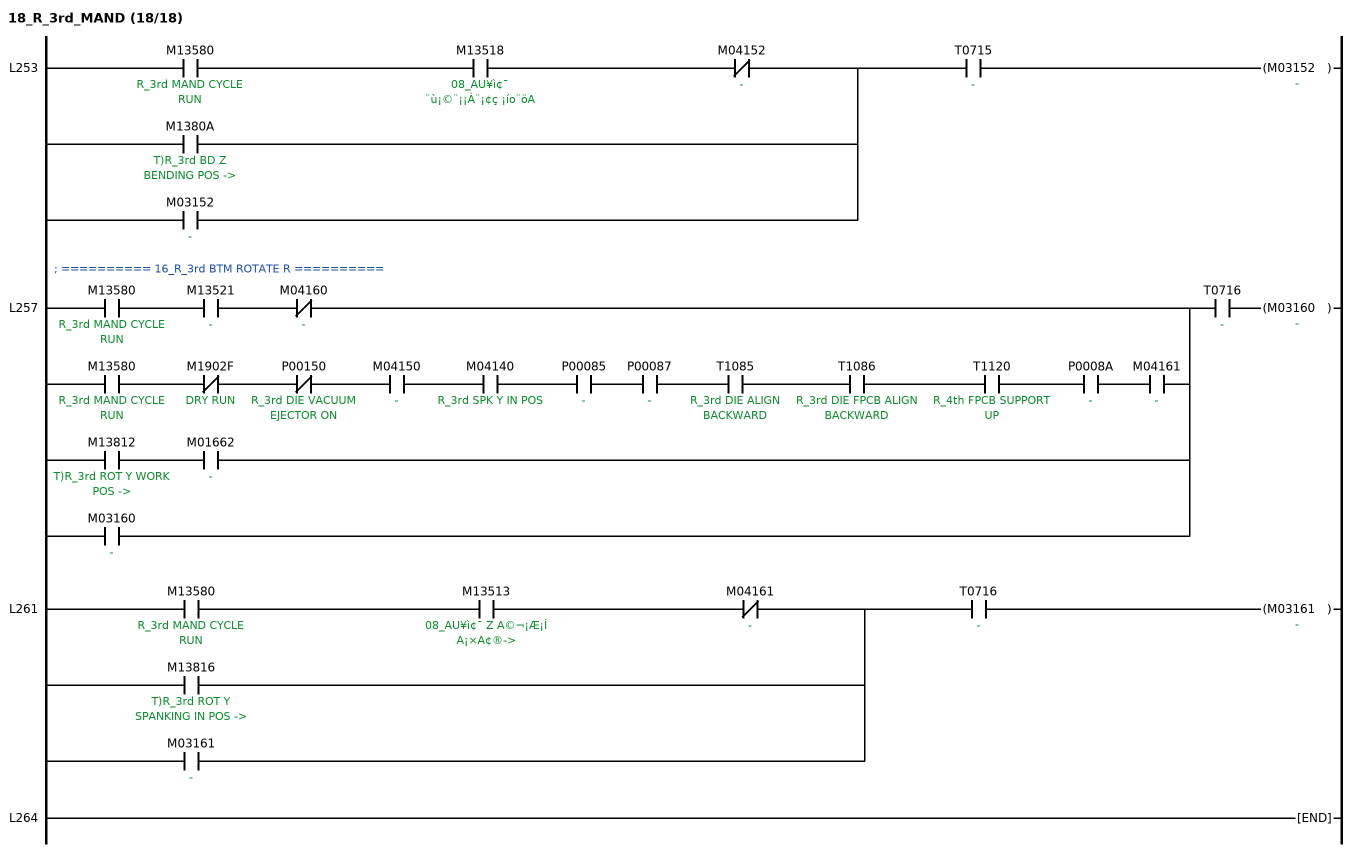
[picture p168: 18_R_3rd_MAND rungs L253-L264]
; L253
LOAD      M13580	// R_3rd MAND CYCLE RUN
AND       M13518	// 08_AU¥ì¢¯ ¨ù¡©¨¡¡À¨¡¢ç ¡ío¨öA
AND NOT   M04152	// -
OR        M1380A	// T)R_3rd BD Z BENDING POS ->
OR        M03152	// -
AND       T0715	// -
OUT       M03152	// -
// ========== 16_R_3rd BTM ROTATE R ==========
; L257
LOAD      M13580	// R_3rd MAND CYCLE RUN
AND       M13521	// -
AND NOT   M04160	// -
LOAD      M13580	// R_3rd MAND CYCLE RUN
AND NOT   M1902F	// DRY RUN
AND NOT   P00150	// R_3rd DIE VACUUM EJECTOR ON
AND       M04150	// -
AND       M04140	// R_3rd SPK Y IN POS
AND       P00085	// -
AND       P00087	// -
AND       T1085	// R_3rd DIE ALIGN BACKWARD
AND       T1086	// R_3rd DIE FPCB ALIGN BACKWARD
AND       T1120	// R_4th FPCB SUPPORT UP
AND       P0008A	// -
AND       M04161	// -
OR LOAD
LOAD      M13812	// T)R_3rd ROT Y WORK POS ->
AND       M01662	// -
OR LOAD
OR        M03160	// -
AND       T0716	// -
OUT       M03160	// -
; L261
LOAD      M13580	// R_3rd MAND CYCLE RUN
AND       M13513	// 08_AU¥ì¢¯ Z A©¬¡Æ¡Ì A¡×A¢®->
AND NOT   M04161	// -
OR        M13816	// T)R_3rd ROT Y SPANKING IN POS ->
OR        M03161	// -
AND       T0716	// -
OUT       M03161	// -
; L264
END

PROGRAM 19_R_TOOL (task: ¨ö¨¬A¥ì CA¡¤I¡¾¡¿¡¤¡Í)

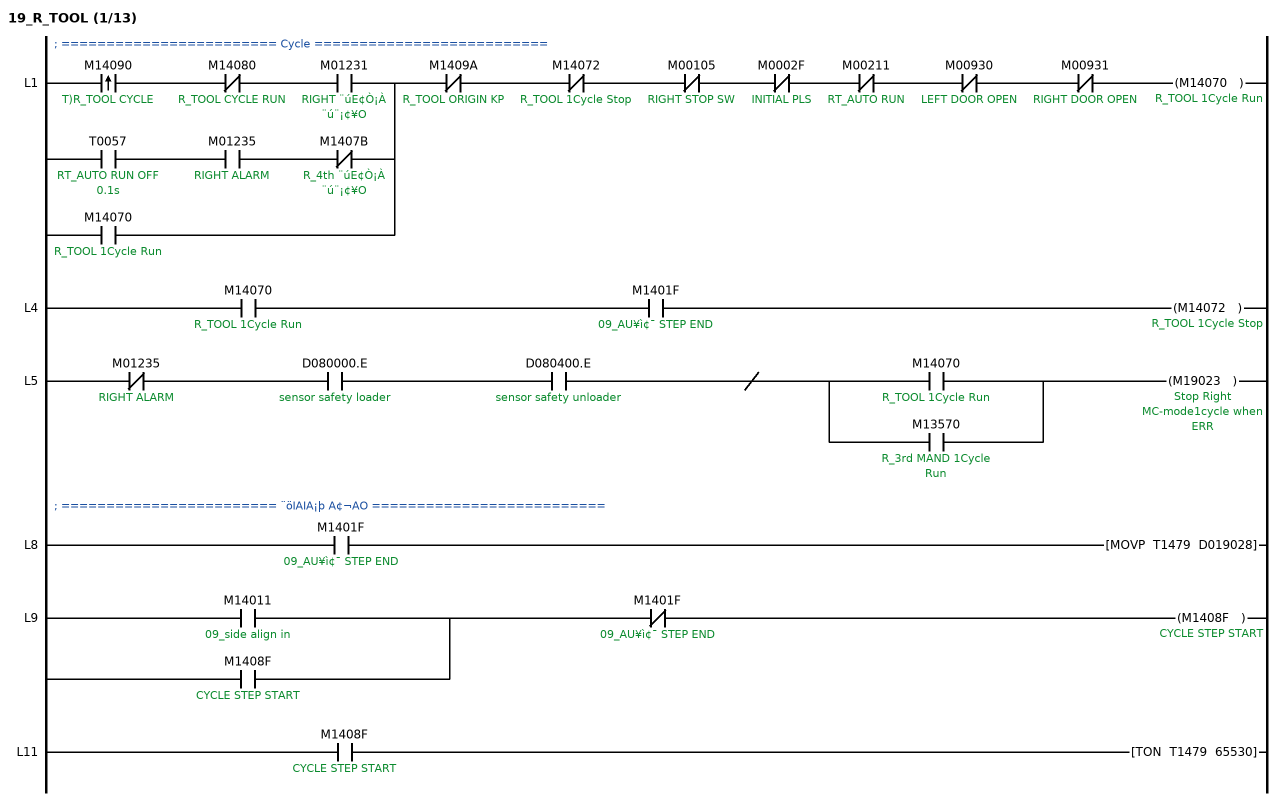
// ======================== Cycle ==========================
; L1
LOADP     M14090	// T)R_TOOL CYCLE
AND NOT   M14080	// R_TOOL CYCLE RUN
AND       M01231	// RIGHT ¨úE¢Ò¡À ¨ú¨¡¢¥O
LOAD      T0057	// RT_AUTO RUN OFF 0.1s
AND       M01235	// RIGHT ALARM
AND NOT   M1407B	// R_4th ¨úE¢Ò¡À ¨ú¨¡¢¥O
OR LOAD
OR        M14070	// R_TOOL 1Cycle Run
AND NOT   M1409A	// R_TOOL ORIGIN KP
AND NOT   M14072	// R_TOOL 1Cycle Stop
AND NOT   M00105	// RIGHT STOP SW
AND NOT   M0002F	// INITIAL PLS
AND NOT   M00211	// RT_AUTO RUN
AND NOT   M00930	// LEFT DOOR OPEN
AND NOT   M00931	// RIGHT DOOR OPEN
OUT       M14070	// R_TOOL 1Cycle Run
; L4
LOAD      M14070	// R_TOOL 1Cycle Run
AND       M1401F	// 09_AU¥ì¢¯ STEP END
OUT       M14072	// R_TOOL 1Cycle Stop
; L5
LOAD NOT  M01235	// RIGHT ALARM
AND       D080000.E	// sensor safety loader
AND       D080400.E	// sensor safety unloader
NOT
LOAD      M14070	// R_TOOL 1Cycle Run
OR        M13570	// R_3rd MAND 1Cycle Run
AND LOAD
OUT       M19023	// Stop Right MC-mode1cycle when ERR
// ======================== ¨öIAIA¡þ A¢¬AO ==========================
; L8
LOAD      M1401F	// 09_AU¥ì¢¯ STEP END
MOVP      T1479 D019028
; L9
LOAD      M14011	// 09_side align in
OR        M1408F	// CYCLE STEP START
AND NOT   M1401F	// 09_AU¥ì¢¯ STEP END
OUT       M1408F	// CYCLE STEP START
; L11
LOAD      M1408F	// CYCLE STEP START
TON       T1479 65530

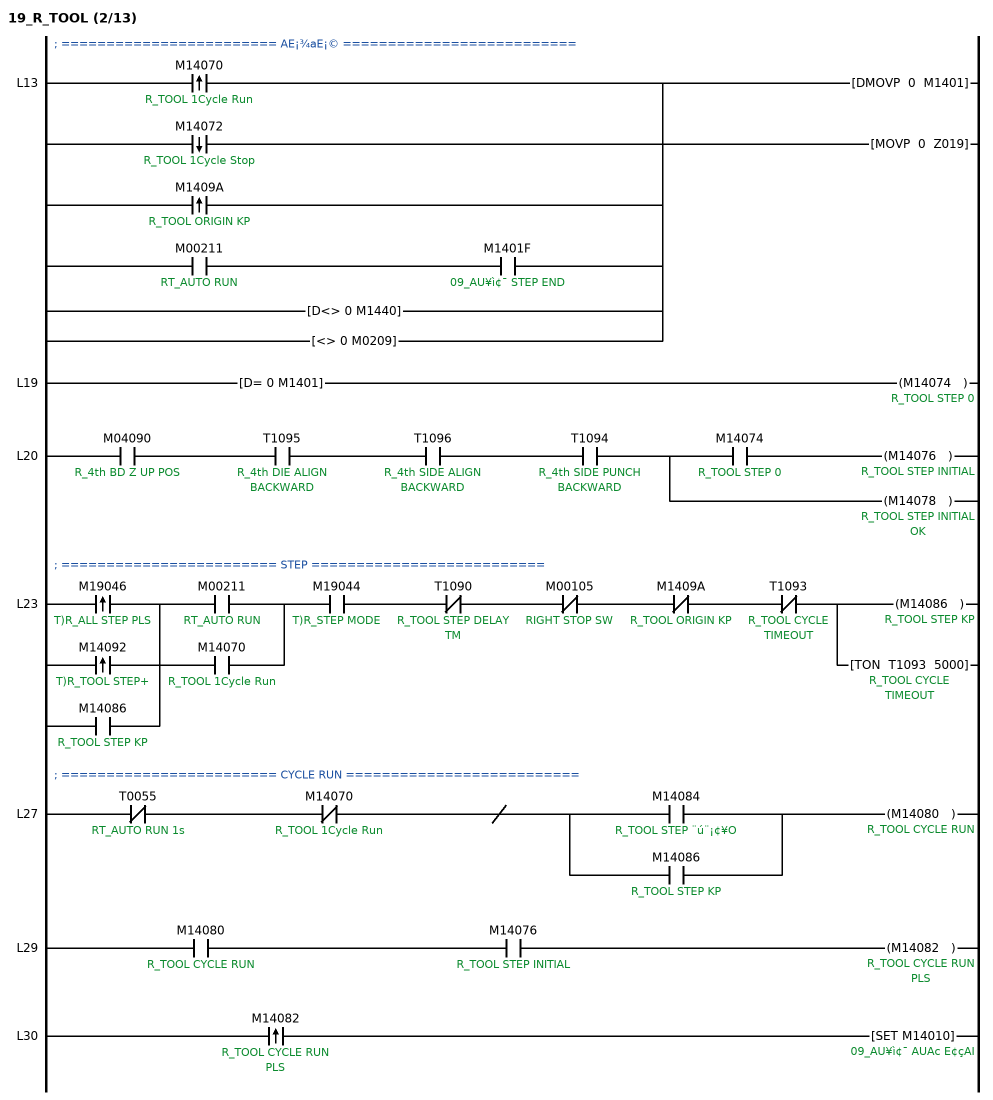
// ======================== AE¡¾aE¡© ==========================
; L13
LOADP     M14070	// R_TOOL 1Cycle Run
ORN       M14072	// R_TOOL 1Cycle Stop
ORP       M1409A	// R_TOOL ORIGIN KP
LOAD      M00211	// RT_AUTO RUN
AND       M1401F	// 09_AU¥ì¢¯ STEP END
OR LOAD
ORD<>     0 M1440
OR<>      0 M0209
DMOVP     0 M1401
MOVP      0 Z019
; L19
LOADD=    0 M1401
OUT       M14074	// R_TOOL STEP 0
; L20
LOAD      M04090	// R_4th BD Z UP POS
AND       T1095	// R_4th DIE ALIGN BACKWARD
AND       T1096	// R_4th SIDE ALIGN BACKWARD
AND       T1094	// R_4th SIDE PUNCH BACKWARD
MPUSH
AND       M14074	// R_TOOL STEP 0
OUT       M14076	// R_TOOL STEP INITIAL
MPOP
OUT       M14078	// R_TOOL STEP INITIAL OK
// ======================== STEP ==========================
; L23
LOADP     M19046	// T)R_ALL STEP PLS
ORP       M14092	// T)R_TOOL STEP+
OR        M14086	// R_TOOL STEP KP
LOAD      M00211	// RT_AUTO RUN
OR        M14070	// R_TOOL 1Cycle Run
AND LOAD
AND       M19044	// T)R_STEP MODE
AND NOT   T1090	// R_TOOL STEP DELAY TM
AND NOT   M00105	// RIGHT STOP SW
AND NOT   M1409A	// R_TOOL ORIGIN KP
AND NOT   T1093	// R_TOOL CYCLE TIMEOUT
OUT       M14086	// R_TOOL STEP KP
TON       T1093 5000	// R_TOOL CYCLE TIMEOUT
// ======================== CYCLE RUN ==========================
; L27
LOAD NOT  T0055	// RT_AUTO RUN 1s
AND NOT   M14070	// R_TOOL 1Cycle Run
NOT
LOAD      M14084	// R_TOOL STEP ¨ú¨¡¢¥O
OR        M14086	// R_TOOL STEP KP
AND LOAD
OUT       M14080	// R_TOOL CYCLE RUN
; L29
LOAD      M14080	// R_TOOL CYCLE RUN
AND       M14076	// R_TOOL STEP INITIAL
OUT       M14082	// R_TOOL CYCLE RUN PLS
; L30
LOADP     M14082	// R_TOOL CYCLE RUN PLS
SET       M14010	// 09_AU¥ì¢¯ AUAc E¢çAI

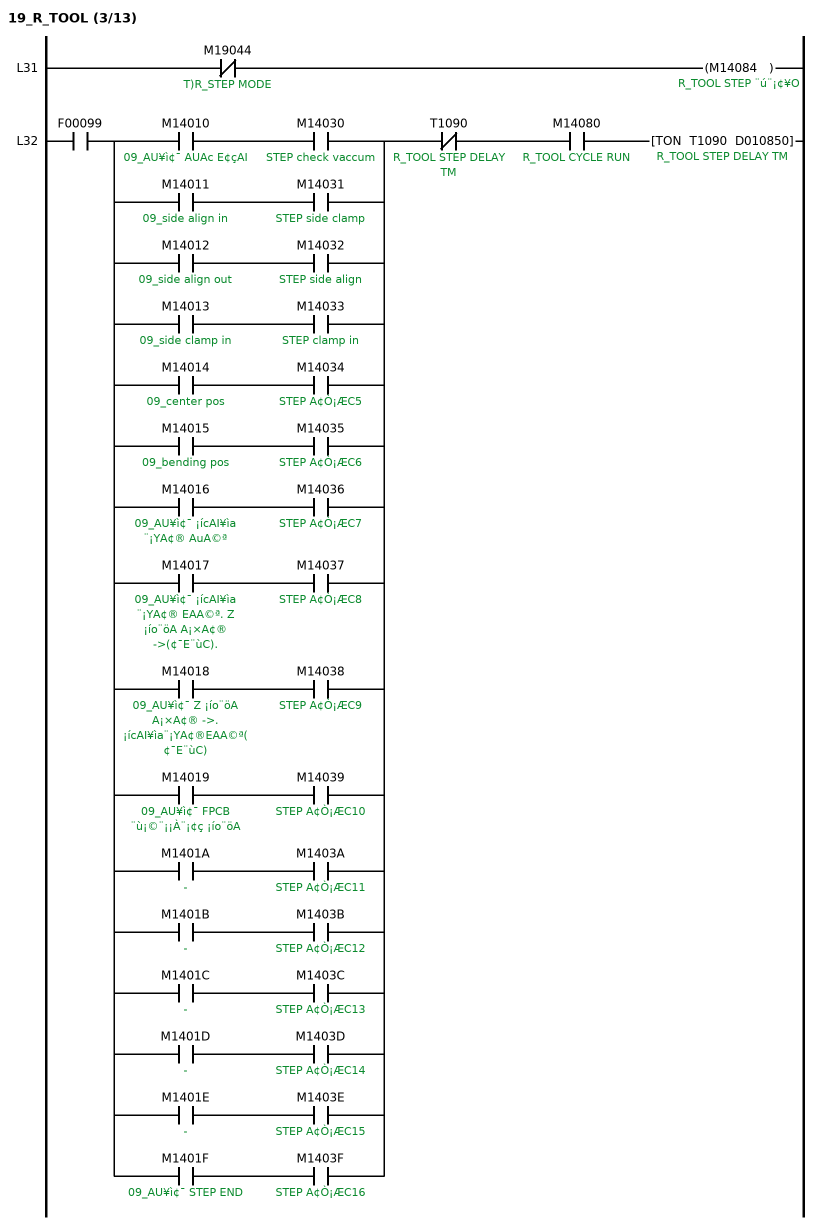
; L31
LOAD NOT  M19044	// T)R_STEP MODE
OUT       M14084	// R_TOOL STEP ¨ú¨¡¢¥O
; L32
LOAD      F00099
LOAD      M14010	// 09_AU¥ì¢¯ AUAc E¢çAI
AND       M14030	// STEP check vaccum
LOAD      M14011	// 09_side align in
AND       M14031	// STEP side clamp
OR LOAD
LOAD      M14012	// 09_side align out
AND       M14032	// STEP side align
OR LOAD
LOAD      M14013	// 09_side clamp in
AND       M14033	// STEP clamp in
OR LOAD
LOAD      M14014	// 09_center pos
AND       M14034	// STEP A¢Ò¡ÆC5
OR LOAD
LOAD      M14015	// 09_bending pos
AND       M14035	// STEP A¢Ò¡ÆC6
OR LOAD
LOAD      M14016	// 09_AU¥ì¢¯ ¡ícAI¥ìa ¨¡YA¢® AuA©ª
AND       M14036	// STEP A¢Ò¡ÆC7
OR LOAD
LOAD      M14017	// 09_AU¥ì¢¯ ¡ícAI¥ìa ¨¡YA¢® EAA©ª. Z ¡ío¨öA A¡×A¢® ->(¢¯E¨ùC).
AND       M14037	// STEP A¢Ò¡ÆC8
OR LOAD
LOAD      M14018	// 09_AU¥ì¢¯ Z ¡ío¨öA A¡×A¢® ->. ¡ícAI¥ìa¨¡YA¢®EAA©ª(¢¯E¨ùC)
AND       M14038	// STEP A¢Ò¡ÆC9
OR LOAD
LOAD      M14019	// 09_AU¥ì¢¯ FPCB ¨ù¡©¨¡¡À¨¡¢ç ¡ío¨öA
AND       M14039	// STEP A¢Ò¡ÆC10
OR LOAD
LOAD      M1401A	// -
AND       M1403A	// STEP A¢Ò¡ÆC11
OR LOAD
LOAD      M1401B	// -
AND       M1403B	// STEP A¢Ò¡ÆC12
OR LOAD
LOAD      M1401C	// -
AND       M1403C	// STEP A¢Ò¡ÆC13
OR LOAD
LOAD      M1401D	// -
AND       M1403D	// STEP A¢Ò¡ÆC14
OR LOAD
LOAD      M1401E	// -
AND       M1403E	// STEP A¢Ò¡ÆC15
OR LOAD
LOAD      M1401F	// 09_AU¥ì¢¯ STEP END
AND       M1403F	// STEP A¢Ò¡ÆC16
OR LOAD
AND LOAD
AND NOT   T1090	// R_TOOL STEP DELAY TM
AND       M14080	// R_TOOL CYCLE RUN
TON       T1090 D010850	// R_TOOL STEP DELAY TM

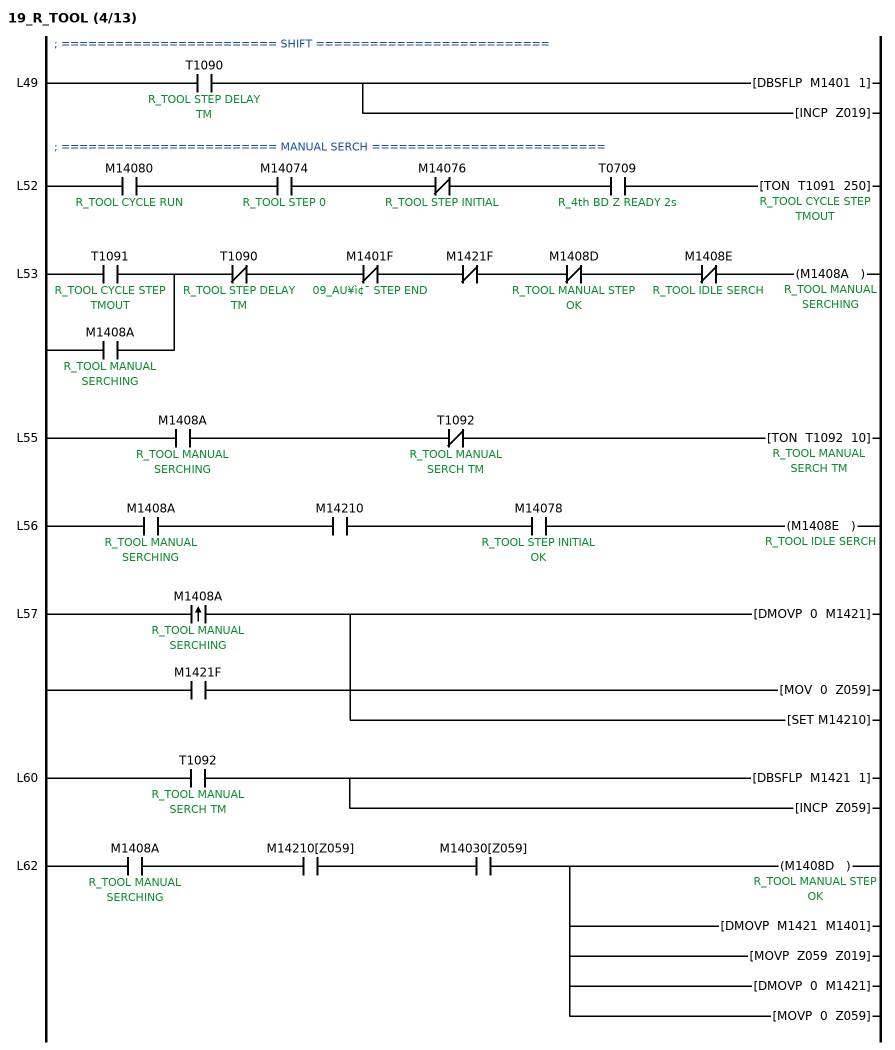
// ======================== SHIFT ==========================
; L49
LOAD      T1090	// R_TOOL STEP DELAY TM
DBSFLP    M1401 1
INCP      Z019
// ======================== MANUAL SERCH ==========================
; L52
LOAD      M14080	// R_TOOL CYCLE RUN
AND       M14074	// R_TOOL STEP 0
AND NOT   M14076	// R_TOOL STEP INITIAL
AND       T0709	// R_4th BD Z READY 2s
TON       T1091 250	// R_TOOL CYCLE STEP TMOUT
; L53
LOAD      T1091	// R_TOOL CYCLE STEP TMOUT
OR        M1408A	// R_TOOL MANUAL SERCHING
AND NOT   T1090	// R_TOOL STEP DELAY TM
AND NOT   M1401F	// 09_AU¥ì¢¯ STEP END
AND NOT   M1421F
AND NOT   M1408D	// R_TOOL MANUAL STEP OK
AND NOT   M1408E	// R_TOOL IDLE SERCH
OUT       M1408A	// R_TOOL MANUAL SERCHING
; L55
LOAD      M1408A	// R_TOOL MANUAL SERCHING
AND NOT   T1092	// R_TOOL MANUAL SERCH TM
TON       T1092 10	// R_TOOL MANUAL SERCH TM
; L56
LOAD      M1408A	// R_TOOL MANUAL SERCHING
AND       M14210
AND       M14078	// R_TOOL STEP INITIAL OK
OUT       M1408E	// R_TOOL IDLE SERCH
; L57
LOADP     M1408A	// R_TOOL MANUAL SERCHING
OR        M1421F
DMOVP     0 M1421
MOV       0 Z059
SET       M14210
; L60
LOAD      T1092	// R_TOOL MANUAL SERCH TM
DBSFLP    M1421 1
INCP      Z059
; L62
LOAD      M1408A	// R_TOOL MANUAL SERCHING
AND       M14210[Z059]
AND       M14030[Z059]
OUT       M1408D	// R_TOOL MANUAL STEP OK
DMOVP     M1421 M1401
MOVP      Z059 Z019
DMOVP     0 M1421
MOVP      0 Z059

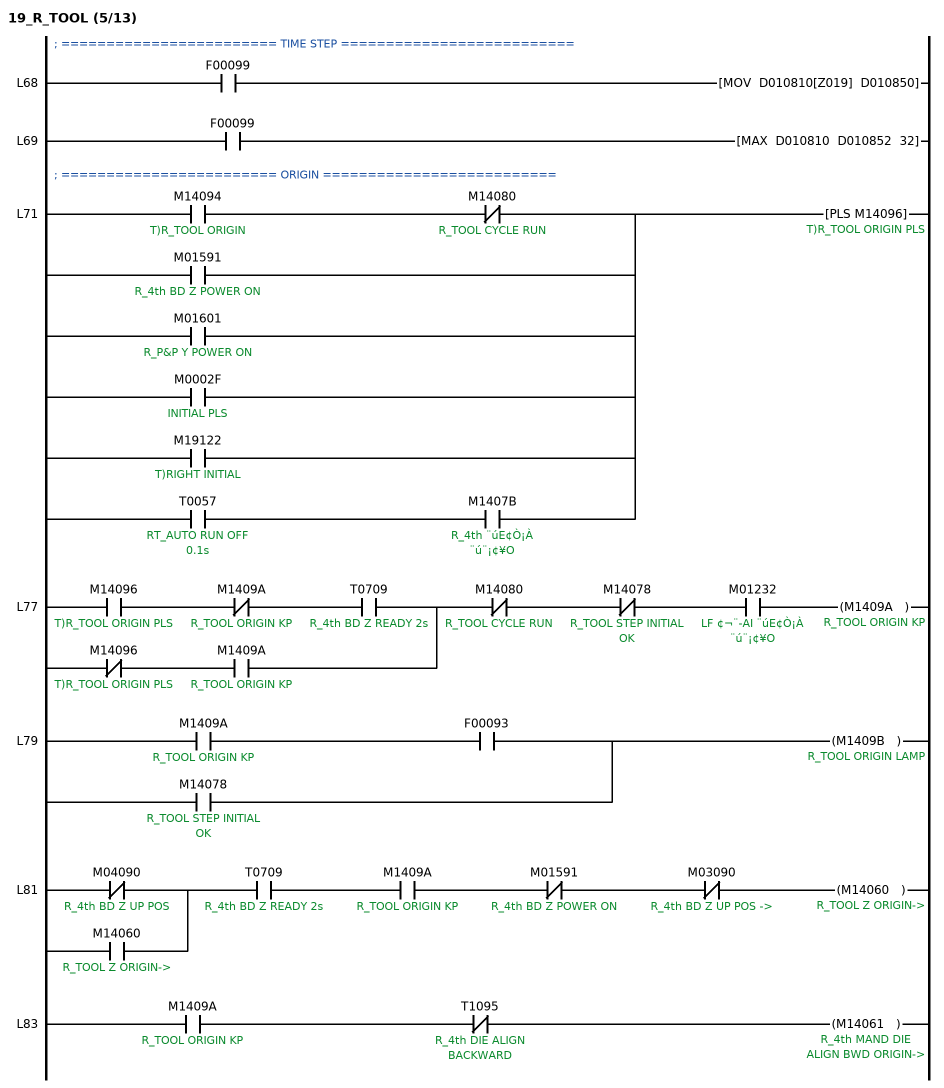
// ======================== TIME STEP ==========================
; L68
LOAD      F00099
MOV       D010810[Z019] D010850
; L69
LOAD      F00099
MAX       D010810 D010852 32
// ======================== ORIGIN ==========================
; L71
LOAD      M14094	// T)R_TOOL ORIGIN
AND NOT   M14080	// R_TOOL CYCLE RUN
OR        M01591	// R_4th BD Z POWER ON
OR        M01601	// R_P&P Y POWER ON
OR        M0002F	// INITIAL PLS
OR        M19122	// T)RIGHT INITIAL
LOAD      T0057	// RT_AUTO RUN OFF 0.1s
AND       M1407B	// R_4th ¨úE¢Ò¡À ¨ú¨¡¢¥O
OR LOAD
OUTP      M14096	// T)R_TOOL ORIGIN PLS
; L77
LOAD      M14096	// T)R_TOOL ORIGIN PLS
AND NOT   M1409A	// R_TOOL ORIGIN KP
AND       T0709	// R_4th BD Z READY 2s
LOAD NOT  M14096	// T)R_TOOL ORIGIN PLS
AND       M1409A	// R_TOOL ORIGIN KP
OR LOAD
AND NOT   M14080	// R_TOOL CYCLE RUN
AND NOT   M14078	// R_TOOL STEP INITIAL OK
AND       M01232	// LF ¢¬¨­AI ¨úE¢Ò¡À ¨ú¨¡¢¥O
OUT       M1409A	// R_TOOL ORIGIN KP
; L79
LOAD      M1409A	// R_TOOL ORIGIN KP
AND       F00093
OR        M14078	// R_TOOL STEP INITIAL OK
OUT       M1409B	// R_TOOL ORIGIN LAMP
; L81
LOAD NOT  M04090	// R_4th BD Z UP POS
OR        M14060	// R_TOOL Z ORIGIN->
AND       T0709	// R_4th BD Z READY 2s
AND       M1409A	// R_TOOL ORIGIN KP
AND NOT   M01591	// R_4th BD Z POWER ON
AND NOT   M03090	// R_4th BD Z UP POS ->
OUT       M14060	// R_TOOL Z ORIGIN->
; L83
LOAD      M1409A	// R_TOOL ORIGIN KP
AND NOT   T1095	// R_4th DIE ALIGN BACKWARD
OUT       M14061	// R_4th MAND DIE ALIGN BWD ORIGIN->

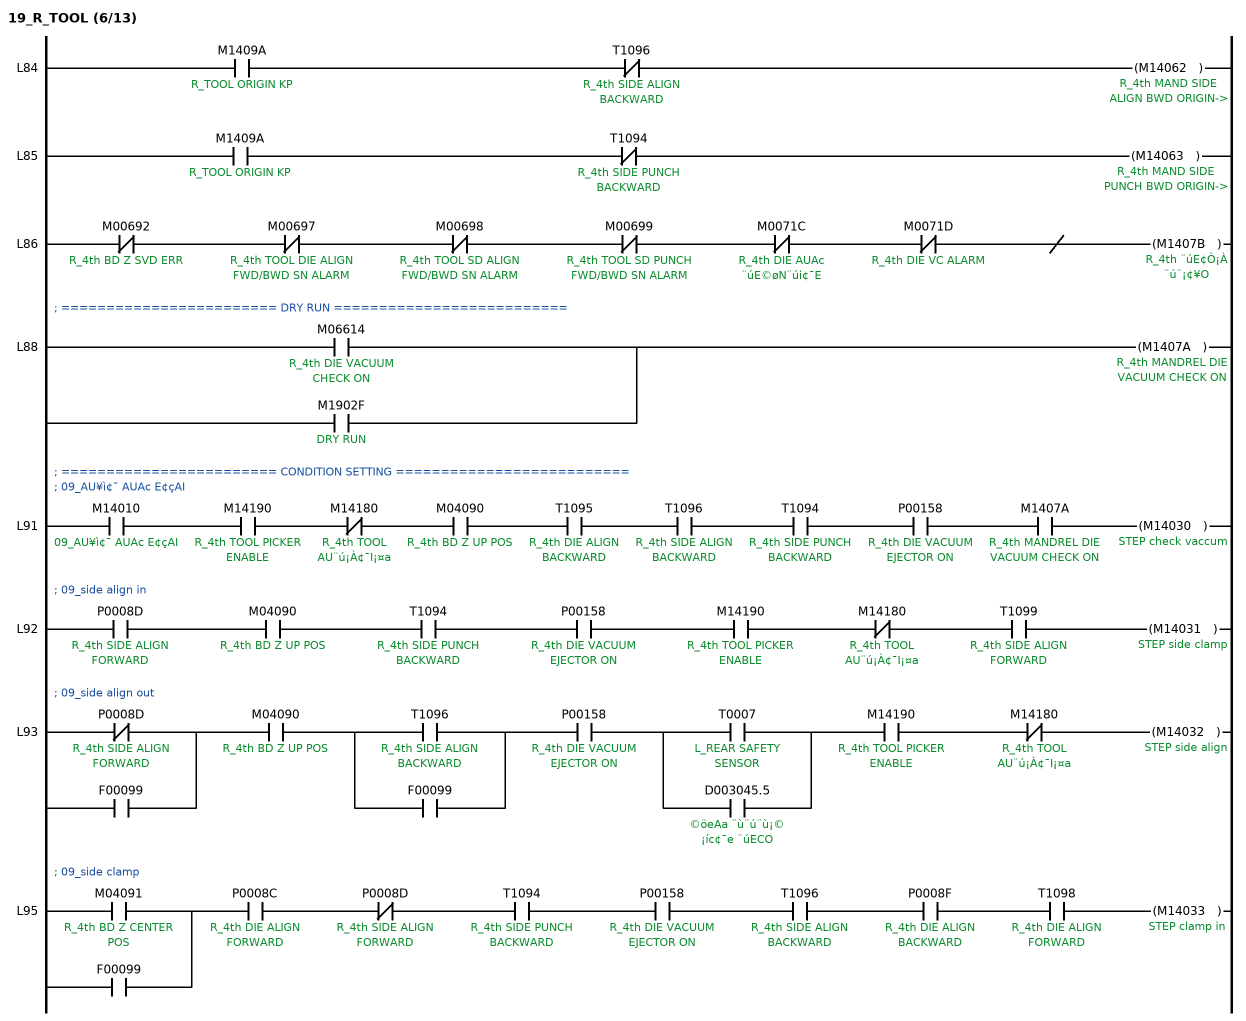
; L84
LOAD      M1409A	// R_TOOL ORIGIN KP
AND NOT   T1096	// R_4th SIDE ALIGN BACKWARD
OUT       M14062	// R_4th MAND SIDE ALIGN BWD ORIGIN->
; L85
LOAD      M1409A	// R_TOOL ORIGIN KP
AND NOT   T1094	// R_4th SIDE PUNCH BACKWARD
OUT       M14063	// R_4th MAND SIDE PUNCH BWD ORIGIN->
; L86
LOAD NOT  M00692	// R_4th BD Z SVD ERR
AND NOT   M00697	// R_4th TOOL DIE ALIGN FWD/BWD SN ALARM
AND NOT   M00698	// R_4th TOOL SD ALIGN FWD/BWD SN ALARM
AND NOT   M00699	// R_4th TOOL SD PUNCH FWD/BWD SN ALARM
AND NOT   M0071C	// R_4th DIE AUAc ¨úE©øN¨úi¢¯E
AND NOT   M0071D	// R_4th DIE VC ALARM
NOT
OUT       M1407B	// R_4th ¨úE¢Ò¡À ¨ú¨¡¢¥O
// ======================== DRY RUN ==========================
; L88
LOAD      M06614	// R_4th DIE VACUUM CHECK ON
OR        M1902F	// DRY RUN
OUT       M1407A	// R_4th MANDREL DIE VACUUM CHECK ON
// ======================== CONDITION SETTING ==========================
; L91
LOAD      M14010	// 09_AU¥ì¢¯ AUAc E¢çAI
AND       M14190	// R_4th TOOL PICKER ENABLE
AND NOT   M14180	// R_4th TOOL AU¨ú¡À¢¯I¡¤a
AND       M04090	// R_4th BD Z UP POS
AND       T1095	// R_4th DIE ALIGN BACKWARD
AND       T1096	// R_4th SIDE ALIGN BACKWARD
AND       T1094	// R_4th SIDE PUNCH BACKWARD
AND       P00158	// R_4th DIE VACUUM EJECTOR ON
AND       M1407A	// R_4th MANDREL DIE VACUUM CHECK ON
OUT       M14030	// STEP check vaccum
// output comment: 09_AU¥ì¢¯ AUAc E¢çAI
; L92
LOAD      P0008D	// R_4th SIDE ALIGN FORWARD
AND       M04090	// R_4th BD Z UP POS
AND       T1094	// R_4th SIDE PUNCH BACKWARD
AND       P00158	// R_4th DIE VACUUM EJECTOR ON
AND       M14190	// R_4th TOOL PICKER ENABLE
AND NOT   M14180	// R_4th TOOL AU¨ú¡À¢¯I¡¤a
AND       T1099	// R_4th SIDE ALIGN FORWARD
OUT       M14031	// STEP side clamp
// output comment: 09_side align in
; L93
LOAD NOT  P0008D	// R_4th SIDE ALIGN FORWARD
OR        F00099
AND       M04090	// R_4th BD Z UP POS
LOAD      T1096	// R_4th SIDE ALIGN BACKWARD
OR        F00099
AND LOAD
AND       P00158	// R_4th DIE VACUUM EJECTOR ON
LOAD      T0007	// L_REAR SAFETY SENSOR
OR        D003045.5	// ©öeAa ¨ù¨ú¨ù¡© ¡íc¢¯e ¨úECO
AND LOAD
AND       M14190	// R_4th TOOL PICKER ENABLE
AND NOT   M14180	// R_4th TOOL AU¨ú¡À¢¯I¡¤a
OUT       M14032	// STEP side align
// output comment: 09_side align out
; L95
LOAD      M04091	// R_4th BD Z CENTER POS
OR        F00099
AND       P0008C	// R_4th DIE ALIGN FORWARD
AND NOT   P0008D	// R_4th SIDE ALIGN FORWARD
AND       T1094	// R_4th SIDE PUNCH BACKWARD
AND       P00158	// R_4th DIE VACUUM EJECTOR ON
AND       T1096	// R_4th SIDE ALIGN BACKWARD
AND       P0008F	// R_4th DIE ALIGN BACKWARD
AND       T1098	// R_4th DIE ALIGN FORWARD
OUT       M14033	// STEP clamp in
// output comment: 09_side clamp

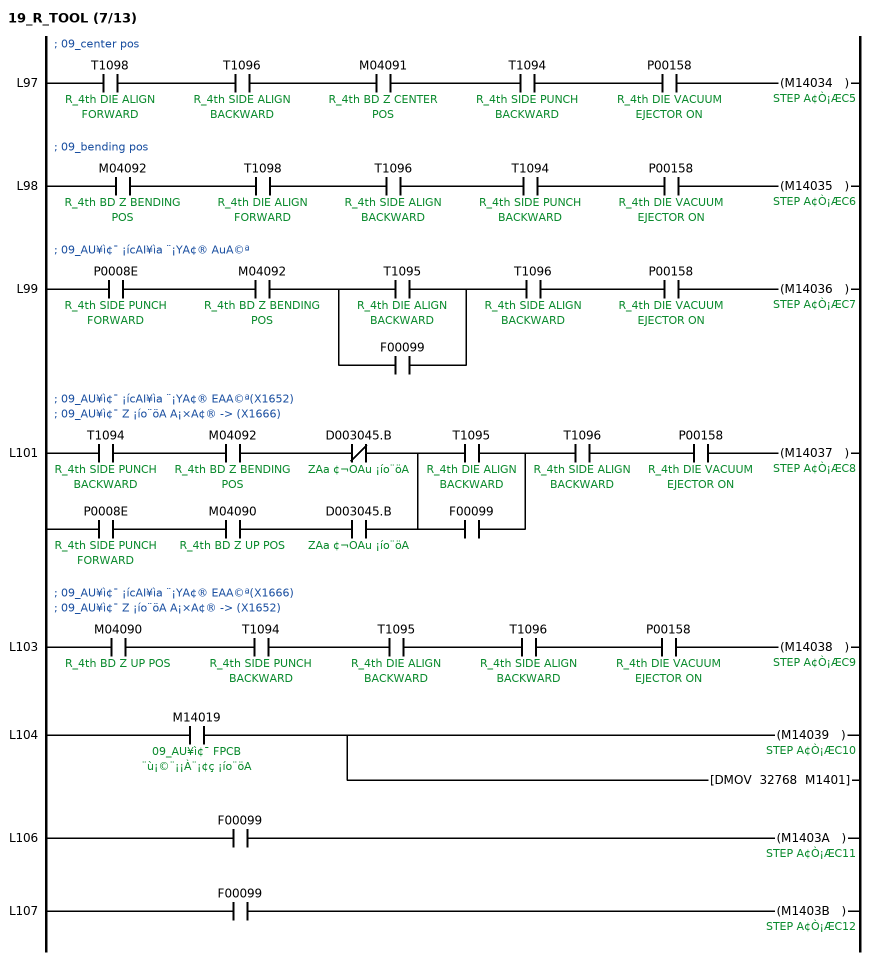
; L97
LOAD      T1098	// R_4th DIE ALIGN FORWARD
AND       T1096	// R_4th SIDE ALIGN BACKWARD
AND       M04091	// R_4th BD Z CENTER POS
AND       T1094	// R_4th SIDE PUNCH BACKWARD
AND       P00158	// R_4th DIE VACUUM EJECTOR ON
OUT       M14034	// STEP A¢Ò¡ÆC5
// output comment: 09_center pos
; L98
LOAD      M04092	// R_4th BD Z BENDING POS
AND       T1098	// R_4th DIE ALIGN FORWARD
AND       T1096	// R_4th SIDE ALIGN BACKWARD
AND       T1094	// R_4th SIDE PUNCH BACKWARD
AND       P00158	// R_4th DIE VACUUM EJECTOR ON
OUT       M14035	// STEP A¢Ò¡ÆC6
// output comment: 09_bending pos
; L99
LOAD      P0008E	// R_4th SIDE PUNCH FORWARD
AND       M04092	// R_4th BD Z BENDING POS
LOAD      T1095	// R_4th DIE ALIGN BACKWARD
OR        F00099
AND LOAD
AND       T1096	// R_4th SIDE ALIGN BACKWARD
AND       P00158	// R_4th DIE VACUUM EJECTOR ON
OUT       M14036	// STEP A¢Ò¡ÆC7
// output comment: 09_AU¥ì¢¯ ¡ícAI¥ìa ¨¡YA¢® AuA©ª
; L101
LOAD      T1094	// R_4th SIDE PUNCH BACKWARD
AND       M04092	// R_4th BD Z BENDING POS
AND NOT   D003045.B	// ZAa ¢¬OAu ¡ío¨öA
LOAD      P0008E	// R_4th SIDE PUNCH FORWARD
AND       M04090	// R_4th BD Z UP POS
AND       D003045.B	// ZAa ¢¬OAu ¡ío¨öA
OR LOAD
LOAD      T1095	// R_4th DIE ALIGN BACKWARD
OR        F00099
AND LOAD
AND       T1096	// R_4th SIDE ALIGN BACKWARD
AND       P00158	// R_4th DIE VACUUM EJECTOR ON
OUT       M14037	// STEP A¢Ò¡ÆC8
// output comment: 09_AU¥ì¢¯ ¡ícAI¥ìa ¨¡YA¢® EAA©ª(X1652) 09_AU¥ì¢¯ Z ¡ío¨öA A¡×A¢® -> (X1666)
; L103
LOAD      M04090	// R_4th BD Z UP POS
AND       T1094	// R_4th SIDE PUNCH BACKWARD
AND       T1095	// R_4th DIE ALIGN BACKWARD
AND       T1096	// R_4th SIDE ALIGN BACKWARD
AND       P00158	// R_4th DIE VACUUM EJECTOR ON
OUT       M14038	// STEP A¢Ò¡ÆC9
// output comment: 09_AU¥ì¢¯ ¡ícAI¥ìa ¨¡YA¢® EAA©ª(X1666) 09_AU¥ì¢¯ Z ¡ío¨öA A¡×A¢® -> (X1652)
; L104
LOAD      M14019	// 09_AU¥ì¢¯ FPCB ¨ù¡©¨¡¡À¨¡¢ç ¡ío¨öA
OUT       M14039	// STEP A¢Ò¡ÆC10
DMOV      32768 M1401
; L106
LOAD      F00099
OUT       M1403A	// STEP A¢Ò¡ÆC11
; L107
LOAD      F00099
OUT       M1403B	// STEP A¢Ò¡ÆC12

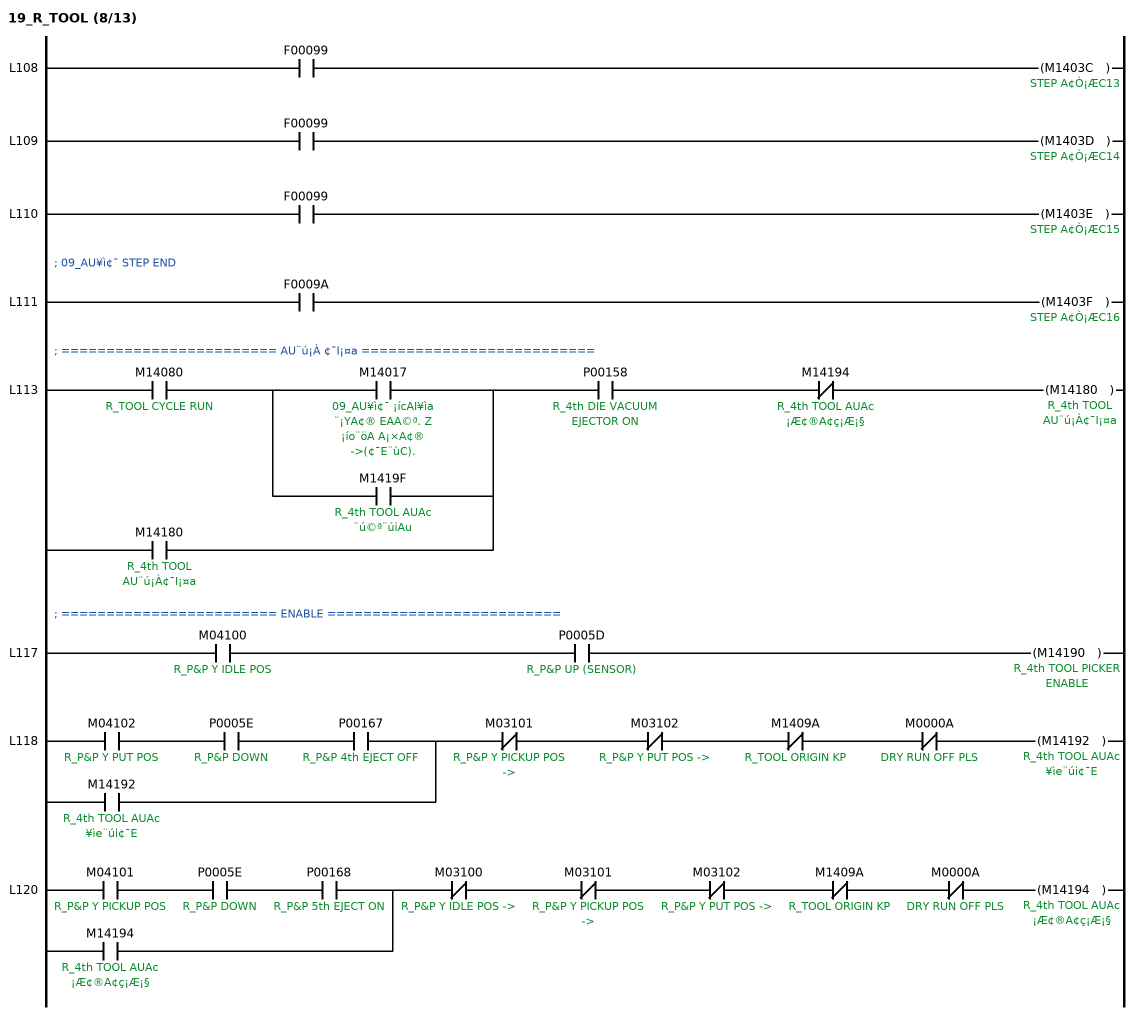
; L108
LOAD      F00099
OUT       M1403C	// STEP A¢Ò¡ÆC13
; L109
LOAD      F00099
OUT       M1403D	// STEP A¢Ò¡ÆC14
; L110
LOAD      F00099
OUT       M1403E	// STEP A¢Ò¡ÆC15
; L111
LOAD      F0009A
OUT       M1403F	// STEP A¢Ò¡ÆC16
// output comment: 09_AU¥ì¢¯ STEP END
// ======================== AU¨ú¡À ¢¯I¡¤a ==========================
; L113
LOAD      M14080	// R_TOOL CYCLE RUN
LOAD      M14017	// 09_AU¥ì¢¯ ¡ícAI¥ìa ¨¡YA¢® EAA©ª. Z ¡ío¨öA A¡×A¢® ->(¢¯E¨ùC).
OR        M1419F	// R_4th TOOL AUAc ¨ú©ª¨úiAu
AND LOAD
OR        M14180	// R_4th TOOL AU¨ú¡À¢¯I¡¤a
AND       P00158	// R_4th DIE VACUUM EJECTOR ON
AND NOT   M14194	// R_4th TOOL AUAc ¡Æ¢®A¢ç¡Æ¡§
OUT       M14180	// R_4th TOOL AU¨ú¡À¢¯I¡¤a
// ======================== ENABLE ==========================
; L117
LOAD      M04100	// R_P&P Y IDLE POS
AND       P0005D	// R_P&P UP (SENSOR)
OUT       M14190	// R_4th TOOL PICKER ENABLE
; L118
LOAD      M04102	// R_P&P Y PUT POS
AND       P0005E	// R_P&P DOWN
AND       P00167	// R_P&P 4th EJECT OFF
OR        M14192	// R_4th TOOL AUAc ¥ìe¨úi¢¯E
AND NOT   M03101	// R_P&P Y PICKUP POS ->
AND NOT   M03102	// R_P&P Y PUT POS ->
AND NOT   M1409A	// R_TOOL ORIGIN KP
AND NOT   M0000A	// DRY RUN OFF PLS
OUT       M14192	// R_4th TOOL AUAc ¥ìe¨úi¢¯E
; L120
LOAD      M04101	// R_P&P Y PICKUP POS
AND       P0005E	// R_P&P DOWN
AND       P00168	// R_P&P 5th EJECT ON
OR        M14194	// R_4th TOOL AUAc ¡Æ¢®A¢ç¡Æ¡§
AND NOT   M03100	// R_P&P Y IDLE POS ->
AND NOT   M03101	// R_P&P Y PICKUP POS ->
AND NOT   M03102	// R_P&P Y PUT POS ->
AND NOT   M1409A	// R_TOOL ORIGIN KP
AND NOT   M0000A	// DRY RUN OFF PLS
OUT       M14194	// R_4th TOOL AUAc ¡Æ¢®A¢ç¡Æ¡§

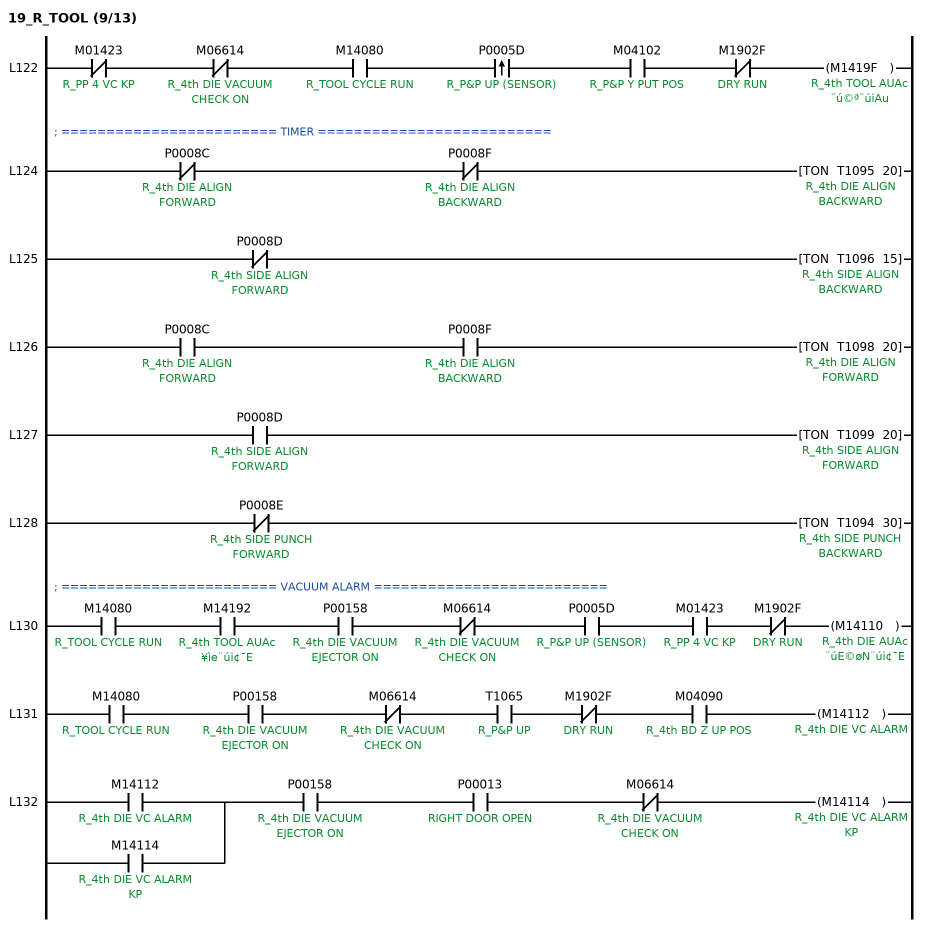
; L122
LOAD NOT  M01423	// R_PP 4 VC KP
AND NOT   M06614	// R_4th DIE VACUUM CHECK ON
AND       M14080	// R_TOOL CYCLE RUN
ANDP      P0005D	// R_P&P UP (SENSOR)
AND       M04102	// R_P&P Y PUT POS
AND NOT   M1902F	// DRY RUN
OUT       M1419F	// R_4th TOOL AUAc ¨ú©ª¨úiAu
// ======================== TIMER ==========================
; L124
LOAD NOT  P0008C	// R_4th DIE ALIGN FORWARD
AND NOT   P0008F	// R_4th DIE ALIGN BACKWARD
TON       T1095 20	// R_4th DIE ALIGN BACKWARD
; L125
LOAD NOT  P0008D	// R_4th SIDE ALIGN FORWARD
TON       T1096 15	// R_4th SIDE ALIGN BACKWARD
; L126
LOAD      P0008C	// R_4th DIE ALIGN FORWARD
AND       P0008F	// R_4th DIE ALIGN BACKWARD
TON       T1098 20	// R_4th DIE ALIGN FORWARD
; L127
LOAD      P0008D	// R_4th SIDE ALIGN FORWARD
TON       T1099 20	// R_4th SIDE ALIGN FORWARD
; L128
LOAD NOT  P0008E	// R_4th SIDE PUNCH FORWARD
TON       T1094 30	// R_4th SIDE PUNCH BACKWARD
// ======================== VACUUM ALARM ==========================
; L130
LOAD      M14080	// R_TOOL CYCLE RUN
AND       M14192	// R_4th TOOL AUAc ¥ìe¨úi¢¯E
AND       P00158	// R_4th DIE VACUUM EJECTOR ON
AND NOT   M06614	// R_4th DIE VACUUM CHECK ON
AND       P0005D	// R_P&P UP (SENSOR)
AND       M01423	// R_PP 4 VC KP
AND NOT   M1902F	// DRY RUN
OUT       M14110	// R_4th DIE AUAc ¨úE©øN¨úi¢¯E
; L131
LOAD      M14080	// R_TOOL CYCLE RUN
AND       P00158	// R_4th DIE VACUUM EJECTOR ON
AND NOT   M06614	// R_4th DIE VACUUM CHECK ON
AND       T1065	// R_P&P UP
AND NOT   M1902F	// DRY RUN
AND       M04090	// R_4th BD Z UP POS
OUT       M14112	// R_4th DIE VC ALARM
; L132
LOAD      M14112	// R_4th DIE VC ALARM
OR        M14114	// R_4th DIE VC ALARM KP
AND       P00158	// R_4th DIE VACUUM EJECTOR ON
AND       P00013	// RIGHT DOOR OPEN
AND NOT   M06614	// R_4th DIE VACUUM CHECK ON
OUT       M14114	// R_4th DIE VC ALARM KP

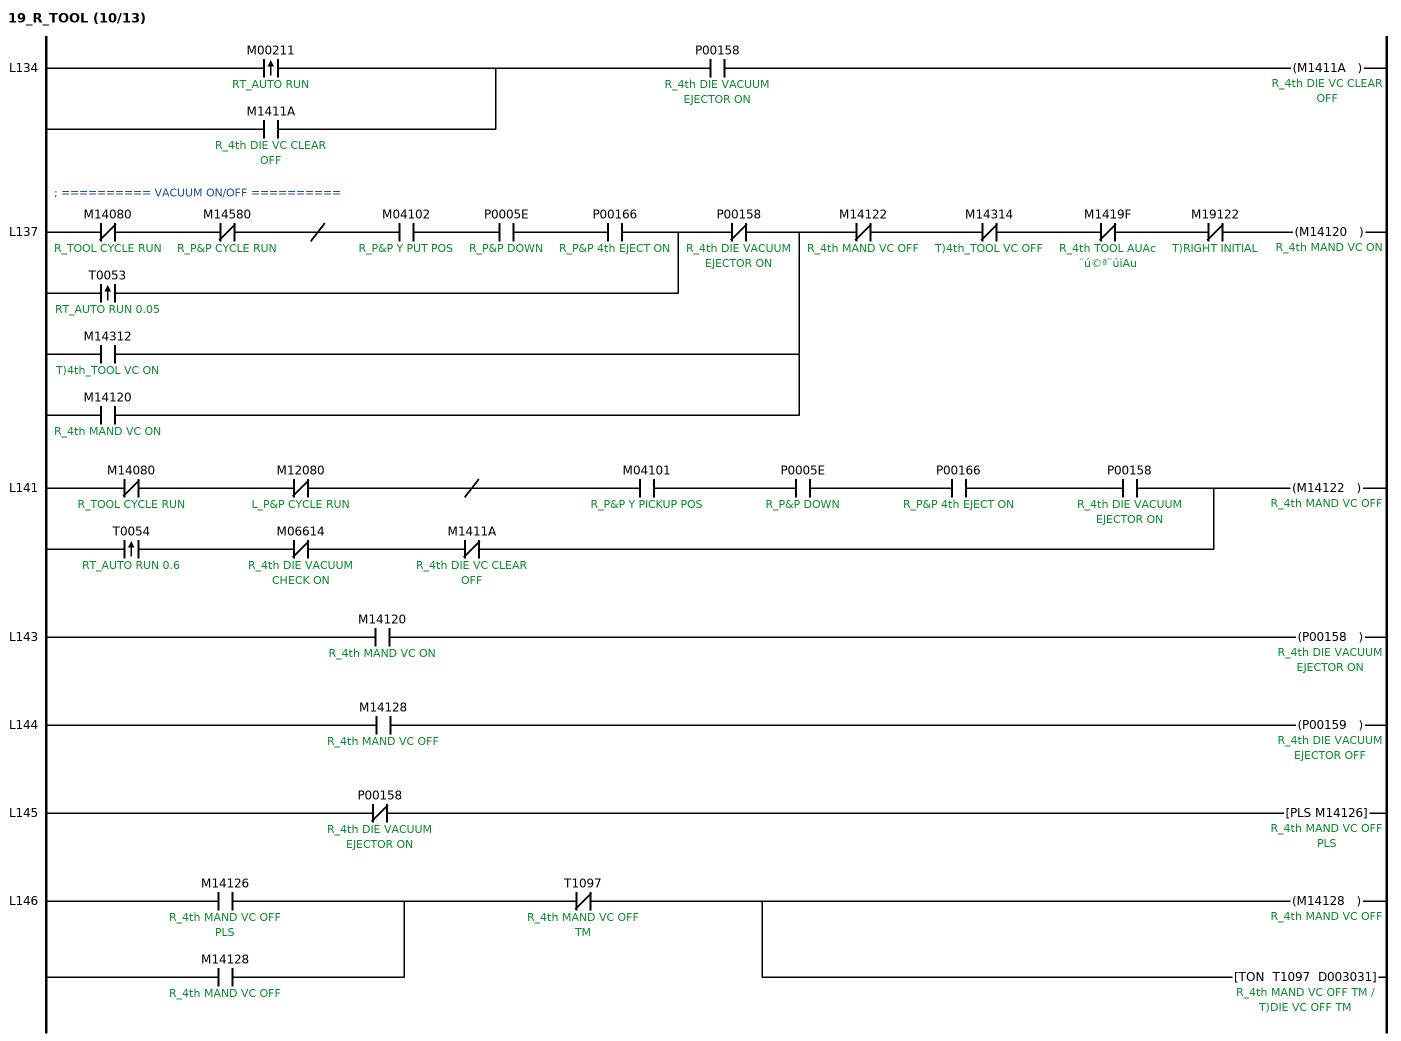
; L134
LOADP     M00211	// RT_AUTO RUN
OR        M1411A	// R_4th DIE VC CLEAR OFF
AND       P00158	// R_4th DIE VACUUM EJECTOR ON
OUT       M1411A	// R_4th DIE VC CLEAR OFF
// ========== VACUUM ON/OFF ==========
; L137
LOAD NOT  M14080	// R_TOOL CYCLE RUN
AND NOT   M14580	// R_P&P CYCLE RUN
NOT
AND       M04102	// R_P&P Y PUT POS
AND       P0005E	// R_P&P DOWN
AND       P00166	// R_P&P 4th EJECT ON
ORP       T0053	// RT_AUTO RUN 0.05
AND NOT   P00158	// R_4th DIE VACUUM EJECTOR ON
OR        M14312	// T)4th_TOOL VC ON
OR        M14120	// R_4th MAND VC ON
AND NOT   M14122	// R_4th MAND VC OFF
AND NOT   M14314	// T)4th_TOOL VC OFF
AND NOT   M1419F	// R_4th TOOL AUAc ¨ú©ª¨úiAu
AND NOT   M19122	// T)RIGHT INITIAL
OUT       M14120	// R_4th MAND VC ON
; L141
LOAD NOT  M14080	// R_TOOL CYCLE RUN
AND NOT   M12080	// L_P&P CYCLE RUN
NOT
AND       M04101	// R_P&P Y PICKUP POS
AND       P0005E	// R_P&P DOWN
AND       P00166	// R_P&P 4th EJECT ON
AND       P00158	// R_4th DIE VACUUM EJECTOR ON
LOADP     T0054	// RT_AUTO RUN 0.6
AND NOT   M06614	// R_4th DIE VACUUM CHECK ON
AND NOT   M1411A	// R_4th DIE VC CLEAR OFF
OR LOAD
OUT       M14122	// R_4th MAND VC OFF
; L143
LOAD      M14120	// R_4th MAND VC ON
OUT       P00158	// R_4th DIE VACUUM EJECTOR ON
; L144
LOAD      M14128	// R_4th MAND VC OFF
OUT       P00159	// R_4th DIE VACUUM EJECTOR OFF
; L145
LOAD NOT  P00158	// R_4th DIE VACUUM EJECTOR ON
OUTP      M14126	// R_4th MAND VC OFF PLS
; L146
LOAD      M14126	// R_4th MAND VC OFF PLS
OR        M14128	// R_4th MAND VC OFF
AND NOT   T1097	// R_4th MAND VC OFF TM
OUT       M14128	// R_4th MAND VC OFF
TON       T1097 D003031	// R_4th MAND VC OFF TM / T)DIE VC OFF TM

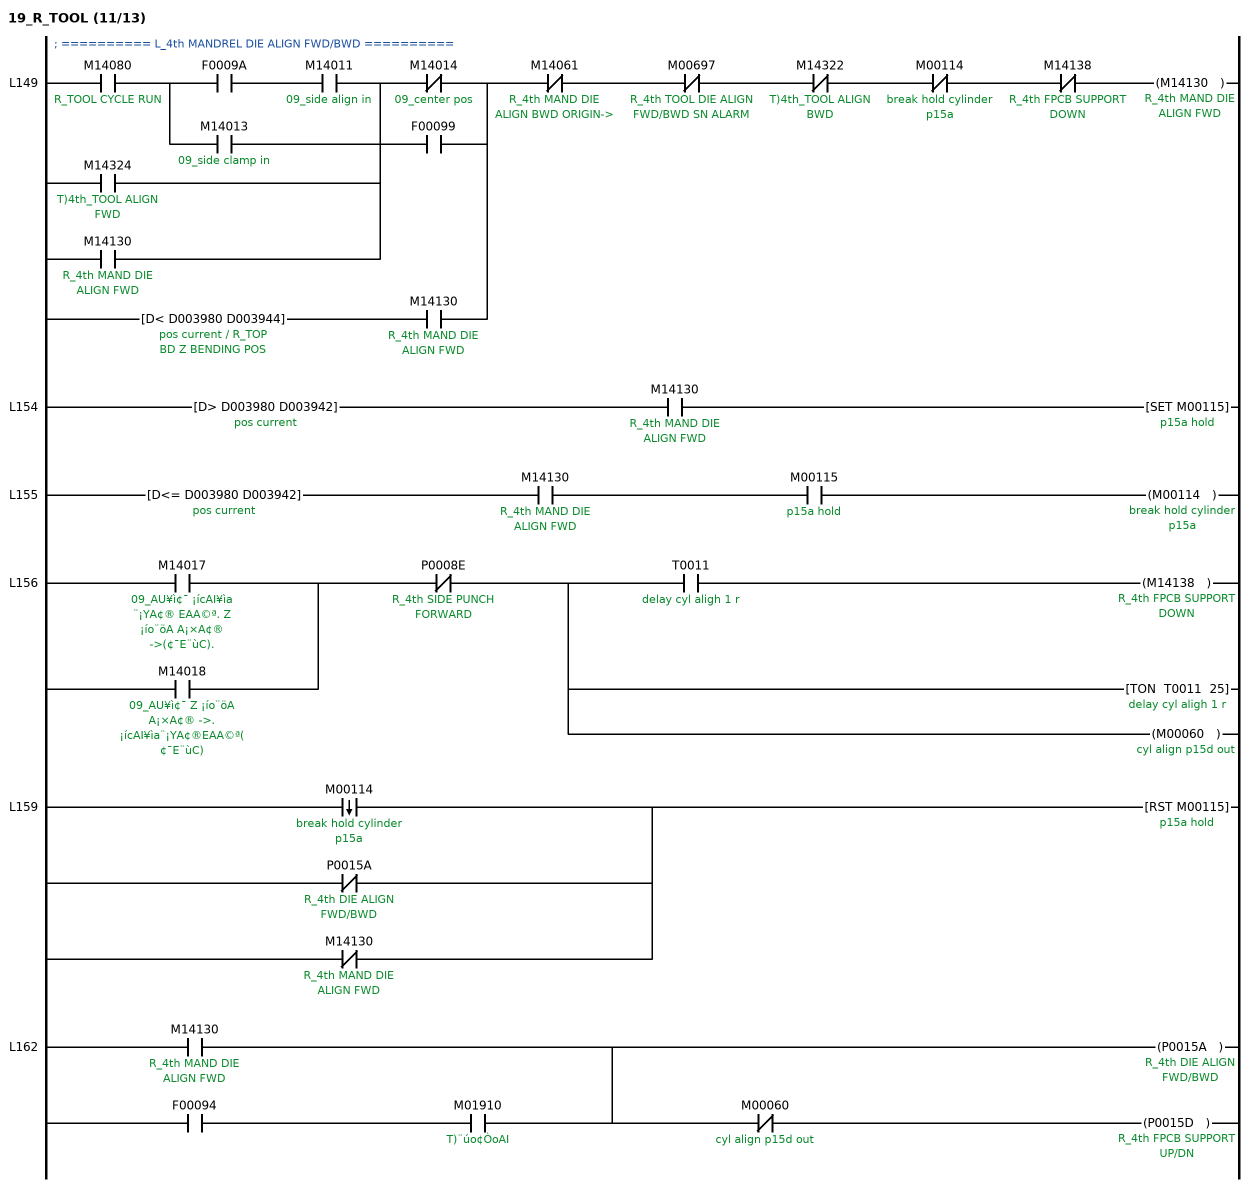
// ========== L_4th MANDREL DIE ALIGN FWD/BWD ==========
; L149
LOAD      M14080	// R_TOOL CYCLE RUN
LOAD      F0009A
AND       M14011	// 09_side align in
OR        M14013	// 09_side clamp in
AND LOAD
OR        M14324	// T)4th_TOOL ALIGN FWD
OR        M14130	// R_4th MAND DIE ALIGN FWD
LOAD NOT  M14014	// 09_center pos
OR        F00099
AND LOAD
LOADD<    D003980 D003944	// pos current / R_TOP BD Z BENDING POS
AND       M14130	// R_4th MAND DIE ALIGN FWD
OR LOAD
AND NOT   M14061	// R_4th MAND DIE ALIGN BWD ORIGIN->
AND NOT   M00697	// R_4th TOOL DIE ALIGN FWD/BWD SN ALARM
AND NOT   M14322	// T)4th_TOOL ALIGN BWD
AND NOT   M00114	// break hold cylinder p15a
AND NOT   M14138	// R_4th FPCB SUPPORT DOWN
OUT       M14130	// R_4th MAND DIE ALIGN FWD
; L154
LOADD>    D003980 D003942	// pos current
AND       M14130	// R_4th MAND DIE ALIGN FWD
SET       M00115	// p15a hold
; L155
LOADD<=   D003980 D003942	// pos current
AND       M14130	// R_4th MAND DIE ALIGN FWD
AND       M00115	// p15a hold
OUT       M00114	// break hold cylinder p15a
; L156
LOAD      M14017	// 09_AU¥ì¢¯ ¡ícAI¥ìa ¨¡YA¢® EAA©ª. Z ¡ío¨öA A¡×A¢® ->(¢¯E¨ùC).
OR        M14018	// 09_AU¥ì¢¯ Z ¡ío¨öA A¡×A¢® ->. ¡ícAI¥ìa¨¡YA¢®EAA©ª(¢¯E¨ùC)
AND NOT   P0008E	// R_4th SIDE PUNCH FORWARD
MPUSH
AND       T0011	// delay cyl aligh 1 r
OUT       M14138	// R_4th FPCB SUPPORT DOWN
MPOP
TON       T0011 25	// delay cyl aligh 1 r
OUT       M00060	// cyl align p15d out
; L159
LOADN     M00114	// break hold cylinder p15a
OR NOT    P0015A	// R_4th DIE ALIGN FWD/BWD
OR NOT    M14130	// R_4th MAND DIE ALIGN FWD
RST       M00115	// p15a hold
; L162
LOAD      M14130	// R_4th MAND DIE ALIGN FWD
LOAD      F00094
AND       M01910	// T)¨úo¢ÒoAI
OR LOAD
OUT       P0015A	// R_4th DIE ALIGN FWD/BWD
AND NOT   M00060	// cyl align p15d out
OUT       P0015D	// R_4th FPCB SUPPORT UP/DN

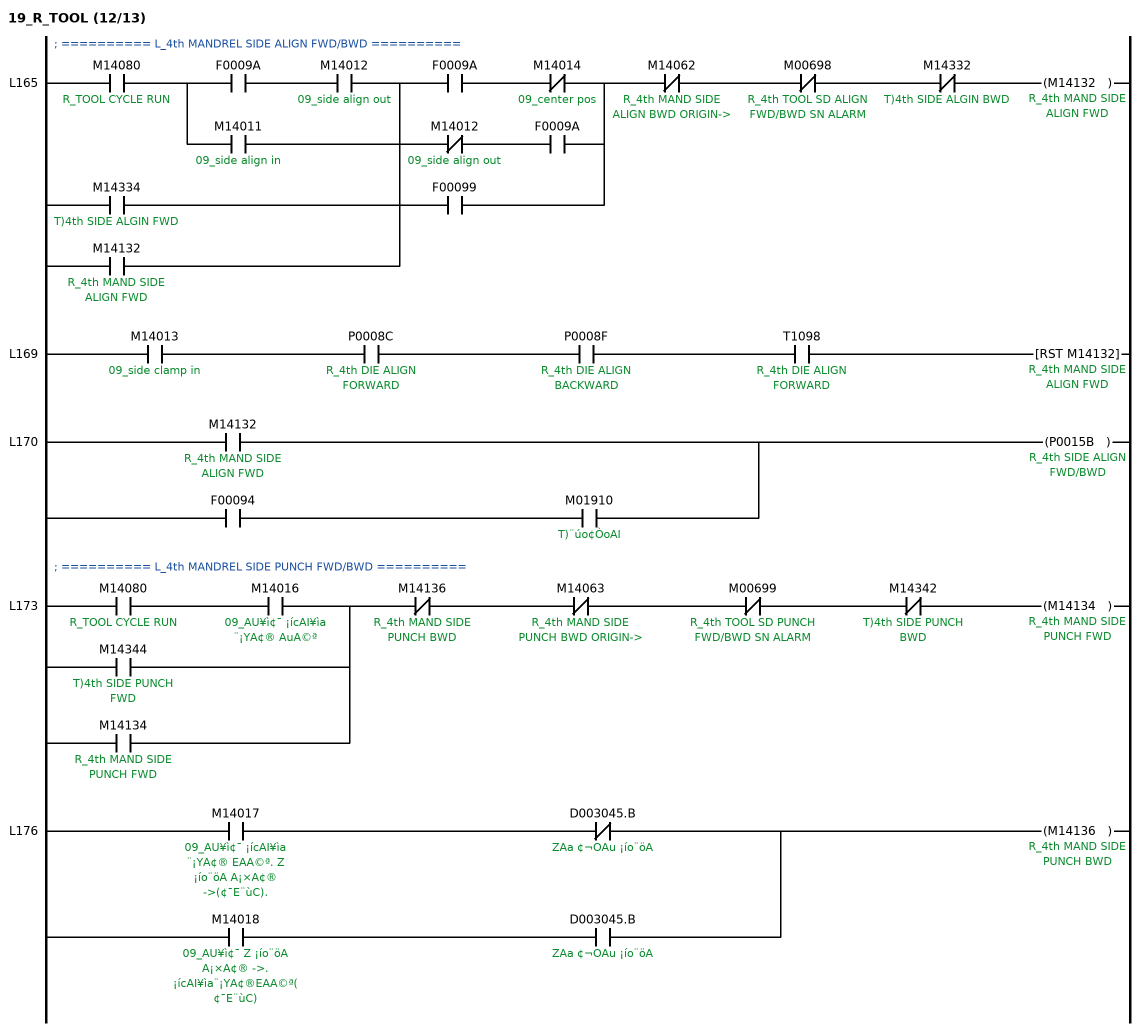
// ========== L_4th MANDREL SIDE ALIGN FWD/BWD ==========
; L165
LOAD      M14080	// R_TOOL CYCLE RUN
LOAD      F0009A
AND       M14012	// 09_side align out
OR        M14011	// 09_side align in
AND LOAD
OR        M14334	// T)4th SIDE ALGIN FWD
OR        M14132	// R_4th MAND SIDE ALIGN FWD
LOAD      F0009A
AND NOT   M14014	// 09_center pos
LOAD NOT  M14012	// 09_side align out
AND       F0009A
OR LOAD
OR        F00099
AND LOAD
AND NOT   M14062	// R_4th MAND SIDE ALIGN BWD ORIGIN->
AND NOT   M00698	// R_4th TOOL SD ALIGN FWD/BWD SN ALARM
AND NOT   M14332	// T)4th SIDE ALGIN BWD
OUT       M14132	// R_4th MAND SIDE ALIGN FWD
; L169
LOAD      M14013	// 09_side clamp in
AND       P0008C	// R_4th DIE ALIGN FORWARD
AND       P0008F	// R_4th DIE ALIGN BACKWARD
AND       T1098	// R_4th DIE ALIGN FORWARD
RST       M14132	// R_4th MAND SIDE ALIGN FWD
; L170
LOAD      M14132	// R_4th MAND SIDE ALIGN FWD
LOAD      F00094
AND       M01910	// T)¨úo¢ÒoAI
OR LOAD
OUT       P0015B	// R_4th SIDE ALIGN FWD/BWD
// ========== L_4th MANDREL SIDE PUNCH FWD/BWD ==========
; L173
LOAD      M14080	// R_TOOL CYCLE RUN
AND       M14016	// 09_AU¥ì¢¯ ¡ícAI¥ìa ¨¡YA¢® AuA©ª
OR        M14344	// T)4th SIDE PUNCH FWD
OR        M14134	// R_4th MAND SIDE PUNCH FWD
AND NOT   M14136	// R_4th MAND SIDE PUNCH BWD
AND NOT   M14063	// R_4th MAND SIDE PUNCH BWD ORIGIN->
AND NOT   M00699	// R_4th TOOL SD PUNCH FWD/BWD SN ALARM
AND NOT   M14342	// T)4th SIDE PUNCH BWD
OUT       M14134	// R_4th MAND SIDE PUNCH FWD
; L176
LOAD      M14017	// 09_AU¥ì¢¯ ¡ícAI¥ìa ¨¡YA¢® EAA©ª. Z ¡ío¨öA A¡×A¢® ->(¢¯E¨ùC).
AND NOT   D003045.B	// ZAa ¢¬OAu ¡ío¨öA
LOAD      M14018	// 09_AU¥ì¢¯ Z ¡ío¨öA A¡×A¢® ->. ¡ícAI¥ìa¨¡YA¢®EAA©ª(¢¯E¨ùC)
AND       D003045.B	// ZAa ¢¬OAu ¡ío¨öA
OR LOAD
OUT       M14136	// R_4th MAND SIDE PUNCH BWD

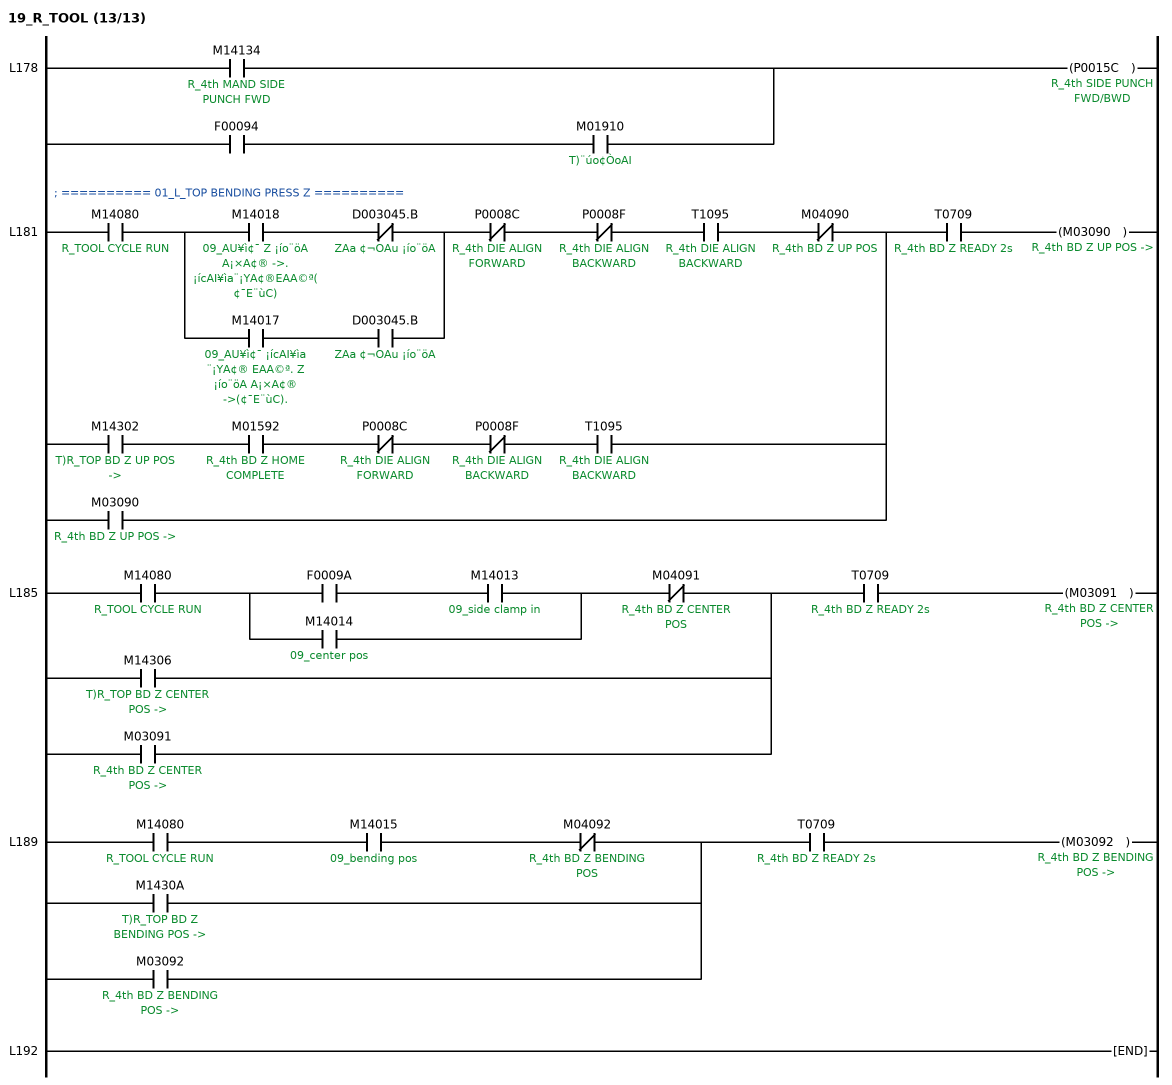
; L178
LOAD      M14134	// R_4th MAND SIDE PUNCH FWD
LOAD      F00094
AND       M01910	// T)¨úo¢ÒoAI
OR LOAD
OUT       P0015C	// R_4th SIDE PUNCH FWD/BWD
// ========== 01_L_TOP BENDING PRESS Z ==========
; L181
LOAD      M14080	// R_TOOL CYCLE RUN
LOAD      M14018	// 09_AU¥ì¢¯ Z ¡ío¨öA A¡×A¢® ->. ¡ícAI¥ìa¨¡YA¢®EAA©ª(¢¯E¨ùC)
AND NOT   D003045.B	// ZAa ¢¬OAu ¡ío¨öA
LOAD      M14017	// 09_AU¥ì¢¯ ¡ícAI¥ìa ¨¡YA¢® EAA©ª. Z ¡ío¨öA A¡×A¢® ->(¢¯E¨ùC).
AND       D003045.B	// ZAa ¢¬OAu ¡ío¨öA
OR LOAD
AND LOAD
AND NOT   P0008C	// R_4th DIE ALIGN FORWARD
AND NOT   P0008F	// R_4th DIE ALIGN BACKWARD
AND       T1095	// R_4th DIE ALIGN BACKWARD
AND NOT   M04090	// R_4th BD Z UP POS
LOAD      M14302	// T)R_TOP BD Z UP POS ->
AND       M01592	// R_4th BD Z HOME COMPLETE
AND NOT   P0008C	// R_4th DIE ALIGN FORWARD
AND NOT   P0008F	// R_4th DIE ALIGN BACKWARD
AND       T1095	// R_4th DIE ALIGN BACKWARD
OR LOAD
OR        M03090	// R_4th BD Z UP POS ->
AND       T0709	// R_4th BD Z READY 2s
OUT       M03090	// R_4th BD Z UP POS ->
; L185
LOAD      M14080	// R_TOOL CYCLE RUN
LOAD      F0009A
AND       M14013	// 09_side clamp in
OR        M14014	// 09_center pos
AND LOAD
AND NOT   M04091	// R_4th BD Z CENTER POS
OR        M14306	// T)R_TOP BD Z CENTER POS ->
OR        M03091	// R_4th BD Z CENTER POS ->
AND       T0709	// R_4th BD Z READY 2s
OUT       M03091	// R_4th BD Z CENTER POS ->
; L189
LOAD      M14080	// R_TOOL CYCLE RUN
AND       M14015	// 09_bending pos
AND NOT   M04092	// R_4th BD Z BENDING POS
OR        M1430A	// T)R_TOP BD Z BENDING POS ->
OR        M03092	// R_4th BD Z BENDING POS ->
AND       T0709	// R_4th BD Z READY 2s
OUT       M03092	// R_4th BD Z BENDING POS ->
; L192
END

PROGRAM 20_R_PP (task: ¨ö¨¬A¥ì CA¡¤I¡¾¡¿¡¤¡Í)

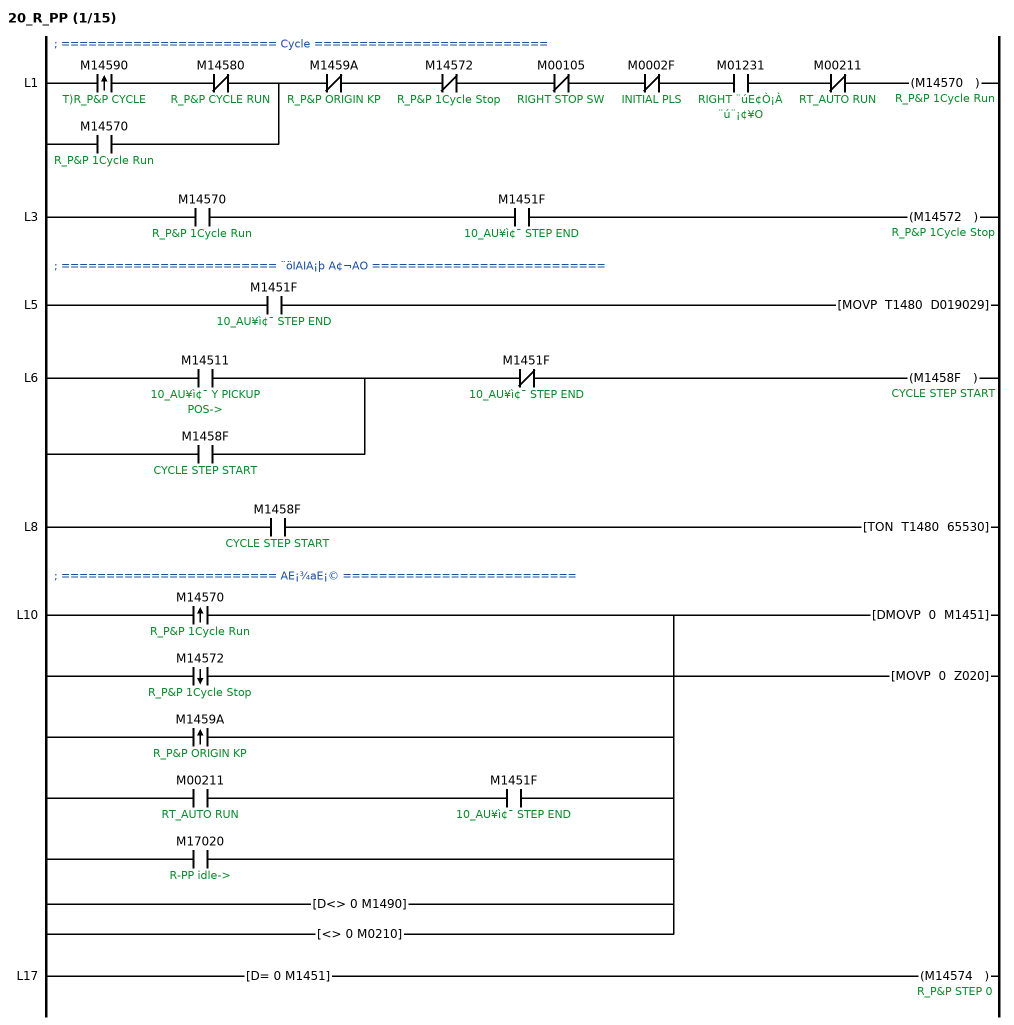
// ======================== Cycle ==========================
; L1
LOADP     M14590	// T)R_P&P CYCLE
AND NOT   M14580	// R_P&P CYCLE RUN
OR        M14570	// R_P&P 1Cycle Run
AND NOT   M1459A	// R_P&P ORIGIN KP
AND NOT   M14572	// R_P&P 1Cycle Stop
AND NOT   M00105	// RIGHT STOP SW
AND NOT   M0002F	// INITIAL PLS
AND       M01231	// RIGHT ¨úE¢Ò¡À ¨ú¨¡¢¥O
AND NOT   M00211	// RT_AUTO RUN
OUT       M14570	// R_P&P 1Cycle Run
; L3
LOAD      M14570	// R_P&P 1Cycle Run
AND       M1451F	// 10_AU¥ì¢¯ STEP END
OUT       M14572	// R_P&P 1Cycle Stop
// ======================== ¨öIAIA¡þ A¢¬AO ==========================
; L5
LOAD      M1451F	// 10_AU¥ì¢¯ STEP END
MOVP      T1480 D019029
; L6
LOAD      M14511	// 10_AU¥ì¢¯ Y PICKUP POS->
OR        M1458F	// CYCLE STEP START
AND NOT   M1451F	// 10_AU¥ì¢¯ STEP END
OUT       M1458F	// CYCLE STEP START
; L8
LOAD      M1458F	// CYCLE STEP START
TON       T1480 65530
// ======================== AE¡¾aE¡© ==========================
; L10
LOADP     M14570	// R_P&P 1Cycle Run
ORN       M14572	// R_P&P 1Cycle Stop
ORP       M1459A	// R_P&P ORIGIN KP
LOAD      M00211	// RT_AUTO RUN
AND       M1451F	// 10_AU¥ì¢¯ STEP END
OR LOAD
OR        M17020	// R-PP idle->
ORD<>     0 M1490
OR<>      0 M0210
DMOVP     0 M1451
MOVP      0 Z020
; L17
LOADD=    0 M1451
OUT       M14574	// R_P&P STEP 0

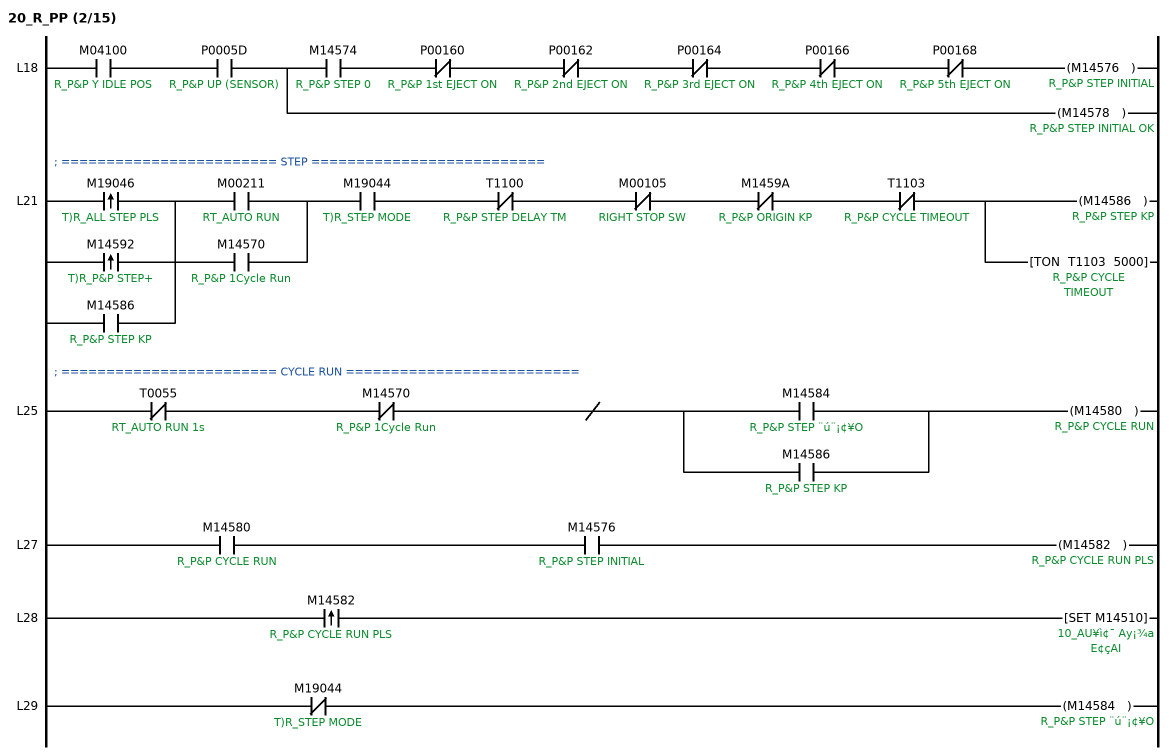
; L18
LOAD      M04100	// R_P&P Y IDLE POS
AND       P0005D	// R_P&P UP (SENSOR)
MPUSH
AND       M14574	// R_P&P STEP 0
AND NOT   P00160	// R_P&P 1st EJECT ON
AND NOT   P00162	// R_P&P 2nd EJECT ON
AND NOT   P00164	// R_P&P 3rd EJECT ON
AND NOT   P00166	// R_P&P 4th EJECT ON
AND NOT   P00168	// R_P&P 5th EJECT ON
OUT       M14576	// R_P&P STEP INITIAL
MPOP
OUT       M14578	// R_P&P STEP INITIAL OK
// ======================== STEP ==========================
; L21
LOADP     M19046	// T)R_ALL STEP PLS
ORP       M14592	// T)R_P&P STEP+
OR        M14586	// R_P&P STEP KP
LOAD      M00211	// RT_AUTO RUN
OR        M14570	// R_P&P 1Cycle Run
AND LOAD
AND       M19044	// T)R_STEP MODE
AND NOT   T1100	// R_P&P STEP DELAY TM
AND NOT   M00105	// RIGHT STOP SW
AND NOT   M1459A	// R_P&P ORIGIN KP
AND NOT   T1103	// R_P&P CYCLE TIMEOUT
OUT       M14586	// R_P&P STEP KP
TON       T1103 5000	// R_P&P CYCLE TIMEOUT
// ======================== CYCLE RUN ==========================
; L25
LOAD NOT  T0055	// RT_AUTO RUN 1s
AND NOT   M14570	// R_P&P 1Cycle Run
NOT
LOAD      M14584	// R_P&P STEP ¨ú¨¡¢¥O
OR        M14586	// R_P&P STEP KP
AND LOAD
OUT       M14580	// R_P&P CYCLE RUN
; L27
LOAD      M14580	// R_P&P CYCLE RUN
AND       M14576	// R_P&P STEP INITIAL
OUT       M14582	// R_P&P CYCLE RUN PLS
; L28
LOADP     M14582	// R_P&P CYCLE RUN PLS
SET       M14510	// 10_AU¥ì¢¯ Ay¡¾a E¢çAI
; L29
LOAD NOT  M19044	// T)R_STEP MODE
OUT       M14584	// R_P&P STEP ¨ú¨¡¢¥O

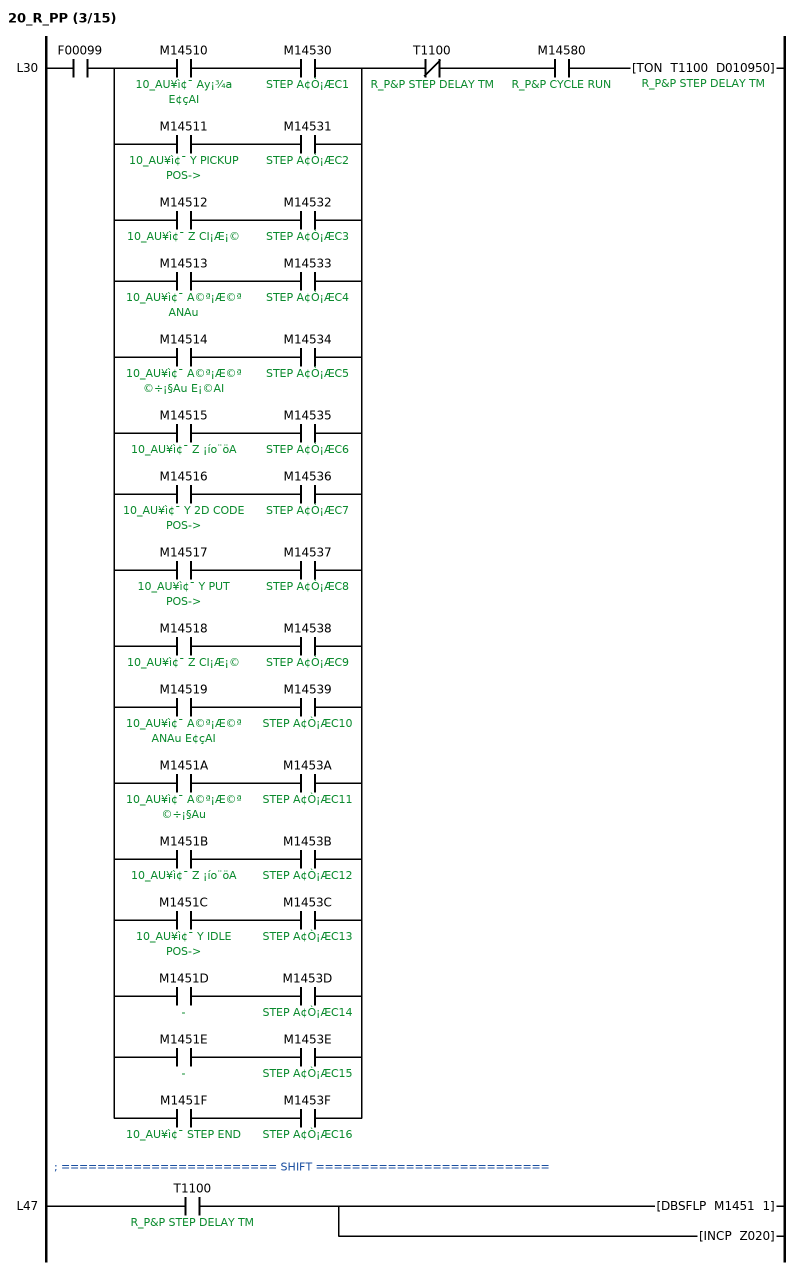
; L30
LOAD      F00099
LOAD      M14510	// 10_AU¥ì¢¯ Ay¡¾a E¢çAI
AND       M14530	// STEP A¢Ò¡ÆC1
LOAD      M14511	// 10_AU¥ì¢¯ Y PICKUP POS->
AND       M14531	// STEP A¢Ò¡ÆC2
OR LOAD
LOAD      M14512	// 10_AU¥ì¢¯ Z CI¡Æ¡©
AND       M14532	// STEP A¢Ò¡ÆC3
OR LOAD
LOAD      M14513	// 10_AU¥ì¢¯ A©ª¡Æ©ª ANAu
AND       M14533	// STEP A¢Ò¡ÆC4
OR LOAD
LOAD      M14514	// 10_AU¥ì¢¯ A©ª¡Æ©ª ©÷¡§Au E¡©AI
AND       M14534	// STEP A¢Ò¡ÆC5
OR LOAD
LOAD      M14515	// 10_AU¥ì¢¯ Z ¡ío¨öA
AND       M14535	// STEP A¢Ò¡ÆC6
OR LOAD
LOAD      M14516	// 10_AU¥ì¢¯ Y 2D CODE POS->
AND       M14536	// STEP A¢Ò¡ÆC7
OR LOAD
LOAD      M14517	// 10_AU¥ì¢¯ Y PUT POS->
AND       M14537	// STEP A¢Ò¡ÆC8
OR LOAD
LOAD      M14518	// 10_AU¥ì¢¯ Z CI¡Æ¡©
AND       M14538	// STEP A¢Ò¡ÆC9
OR LOAD
LOAD      M14519	// 10_AU¥ì¢¯ A©ª¡Æ©ª ANAu E¢çAI
AND       M14539	// STEP A¢Ò¡ÆC10
OR LOAD
LOAD      M1451A	// 10_AU¥ì¢¯ A©ª¡Æ©ª ©÷¡§Au
AND       M1453A	// STEP A¢Ò¡ÆC11
OR LOAD
LOAD      M1451B	// 10_AU¥ì¢¯ Z ¡ío¨öA
AND       M1453B	// STEP A¢Ò¡ÆC12
OR LOAD
LOAD      M1451C	// 10_AU¥ì¢¯ Y IDLE POS->
AND       M1453C	// STEP A¢Ò¡ÆC13
OR LOAD
LOAD      M1451D	// -
AND       M1453D	// STEP A¢Ò¡ÆC14
OR LOAD
LOAD      M1451E	// -
AND       M1453E	// STEP A¢Ò¡ÆC15
OR LOAD
LOAD      M1451F	// 10_AU¥ì¢¯ STEP END
AND       M1453F	// STEP A¢Ò¡ÆC16
OR LOAD
AND LOAD
AND NOT   T1100	// R_P&P STEP DELAY TM
AND       M14580	// R_P&P CYCLE RUN
TON       T1100 D010950	// R_P&P STEP DELAY TM
// ======================== SHIFT ==========================
; L47
LOAD      T1100	// R_P&P STEP DELAY TM
DBSFLP    M1451 1
INCP      Z020

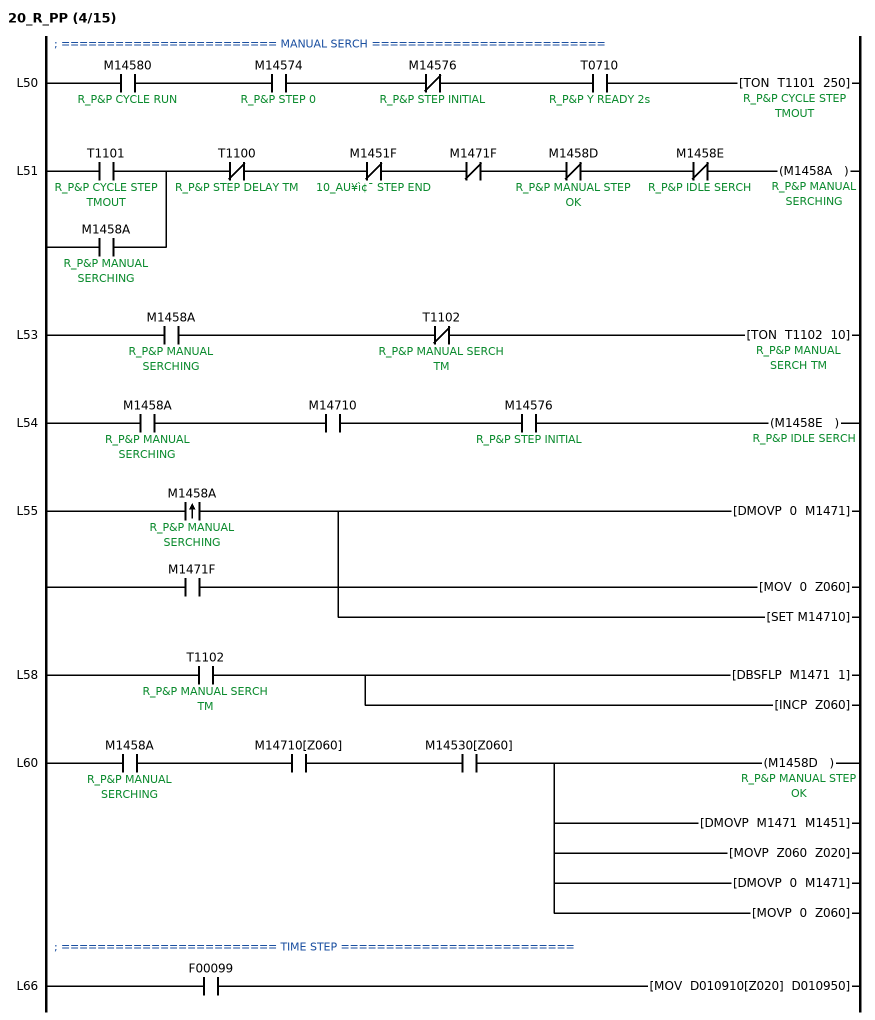
// ======================== MANUAL SERCH ==========================
; L50
LOAD      M14580	// R_P&P CYCLE RUN
AND       M14574	// R_P&P STEP 0
AND NOT   M14576	// R_P&P STEP INITIAL
AND       T0710	// R_P&P Y READY 2s
TON       T1101 250	// R_P&P CYCLE STEP TMOUT
; L51
LOAD      T1101	// R_P&P CYCLE STEP TMOUT
OR        M1458A	// R_P&P MANUAL SERCHING
AND NOT   T1100	// R_P&P STEP DELAY TM
AND NOT   M1451F	// 10_AU¥ì¢¯ STEP END
AND NOT   M1471F
AND NOT   M1458D	// R_P&P MANUAL STEP OK
AND NOT   M1458E	// R_P&P IDLE SERCH
OUT       M1458A	// R_P&P MANUAL SERCHING
; L53
LOAD      M1458A	// R_P&P MANUAL SERCHING
AND NOT   T1102	// R_P&P MANUAL SERCH TM
TON       T1102 10	// R_P&P MANUAL SERCH TM
; L54
LOAD      M1458A	// R_P&P MANUAL SERCHING
AND       M14710
AND       M14576	// R_P&P STEP INITIAL
OUT       M1458E	// R_P&P IDLE SERCH
; L55
LOADP     M1458A	// R_P&P MANUAL SERCHING
OR        M1471F
DMOVP     0 M1471
MOV       0 Z060
SET       M14710
; L58
LOAD      T1102	// R_P&P MANUAL SERCH TM
DBSFLP    M1471 1
INCP      Z060
; L60
LOAD      M1458A	// R_P&P MANUAL SERCHING
AND       M14710[Z060]
AND       M14530[Z060]
OUT       M1458D	// R_P&P MANUAL STEP OK
DMOVP     M1471 M1451
MOVP      Z060 Z020
DMOVP     0 M1471
MOVP      0 Z060
// ======================== TIME STEP ==========================
; L66
LOAD      F00099
MOV       D010910[Z020] D010950

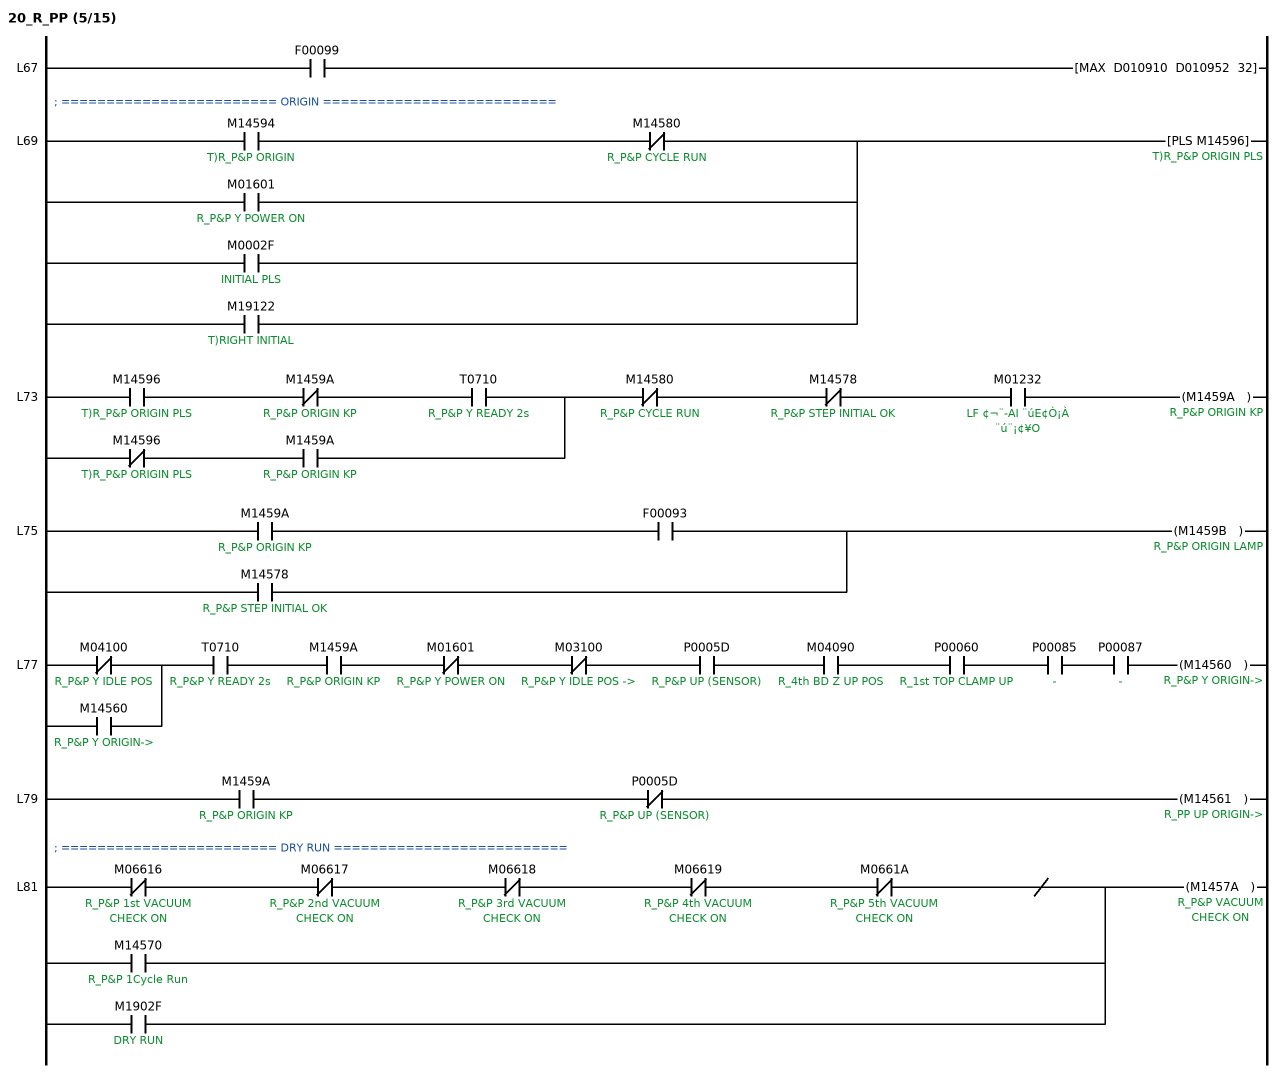
; L67
LOAD      F00099
MAX       D010910 D010952 32
// ======================== ORIGIN ==========================
; L69
LOAD      M14594	// T)R_P&P ORIGIN
AND NOT   M14580	// R_P&P CYCLE RUN
OR        M01601	// R_P&P Y POWER ON
OR        M0002F	// INITIAL PLS
OR        M19122	// T)RIGHT INITIAL
OUTP      M14596	// T)R_P&P ORIGIN PLS
; L73
LOAD      M14596	// T)R_P&P ORIGIN PLS
AND NOT   M1459A	// R_P&P ORIGIN KP
AND       T0710	// R_P&P Y READY 2s
LOAD NOT  M14596	// T)R_P&P ORIGIN PLS
AND       M1459A	// R_P&P ORIGIN KP
OR LOAD
AND NOT   M14580	// R_P&P CYCLE RUN
AND NOT   M14578	// R_P&P STEP INITIAL OK
AND       M01232	// LF ¢¬¨­AI ¨úE¢Ò¡À ¨ú¨¡¢¥O
OUT       M1459A	// R_P&P ORIGIN KP
; L75
LOAD      M1459A	// R_P&P ORIGIN KP
AND       F00093
OR        M14578	// R_P&P STEP INITIAL OK
OUT       M1459B	// R_P&P ORIGIN LAMP
; L77
LOAD NOT  M04100	// R_P&P Y IDLE POS
OR        M14560	// R_P&P Y ORIGIN->
AND       T0710	// R_P&P Y READY 2s
AND       M1459A	// R_P&P ORIGIN KP
AND NOT   M01601	// R_P&P Y POWER ON
AND NOT   M03100	// R_P&P Y IDLE POS ->
AND       P0005D	// R_P&P UP (SENSOR)
AND       M04090	// R_4th BD Z UP POS
AND       P00060	// R_1st TOP CLAMP UP
AND       P00085	// -
AND       P00087	// -
OUT       M14560	// R_P&P Y ORIGIN->
; L79
LOAD      M1459A	// R_P&P ORIGIN KP
AND NOT   P0005D	// R_P&P UP (SENSOR)
OUT       M14561	// R_PP UP ORIGIN->
// ======================== DRY RUN ==========================
; L81
LOAD NOT  M06616	// R_P&P 1st VACUUM CHECK ON
AND NOT   M06617	// R_P&P 2nd VACUUM CHECK ON
AND NOT   M06618	// R_P&P 3rd VACUUM CHECK ON
AND NOT   M06619	// R_P&P 4th VACUUM CHECK ON
AND NOT   M0661A	// R_P&P 5th VACUUM CHECK ON
NOT
OR        M14570	// R_P&P 1Cycle Run
OR        M1902F	// DRY RUN
OUT       M1457A	// R_P&P VACUUM CHECK ON

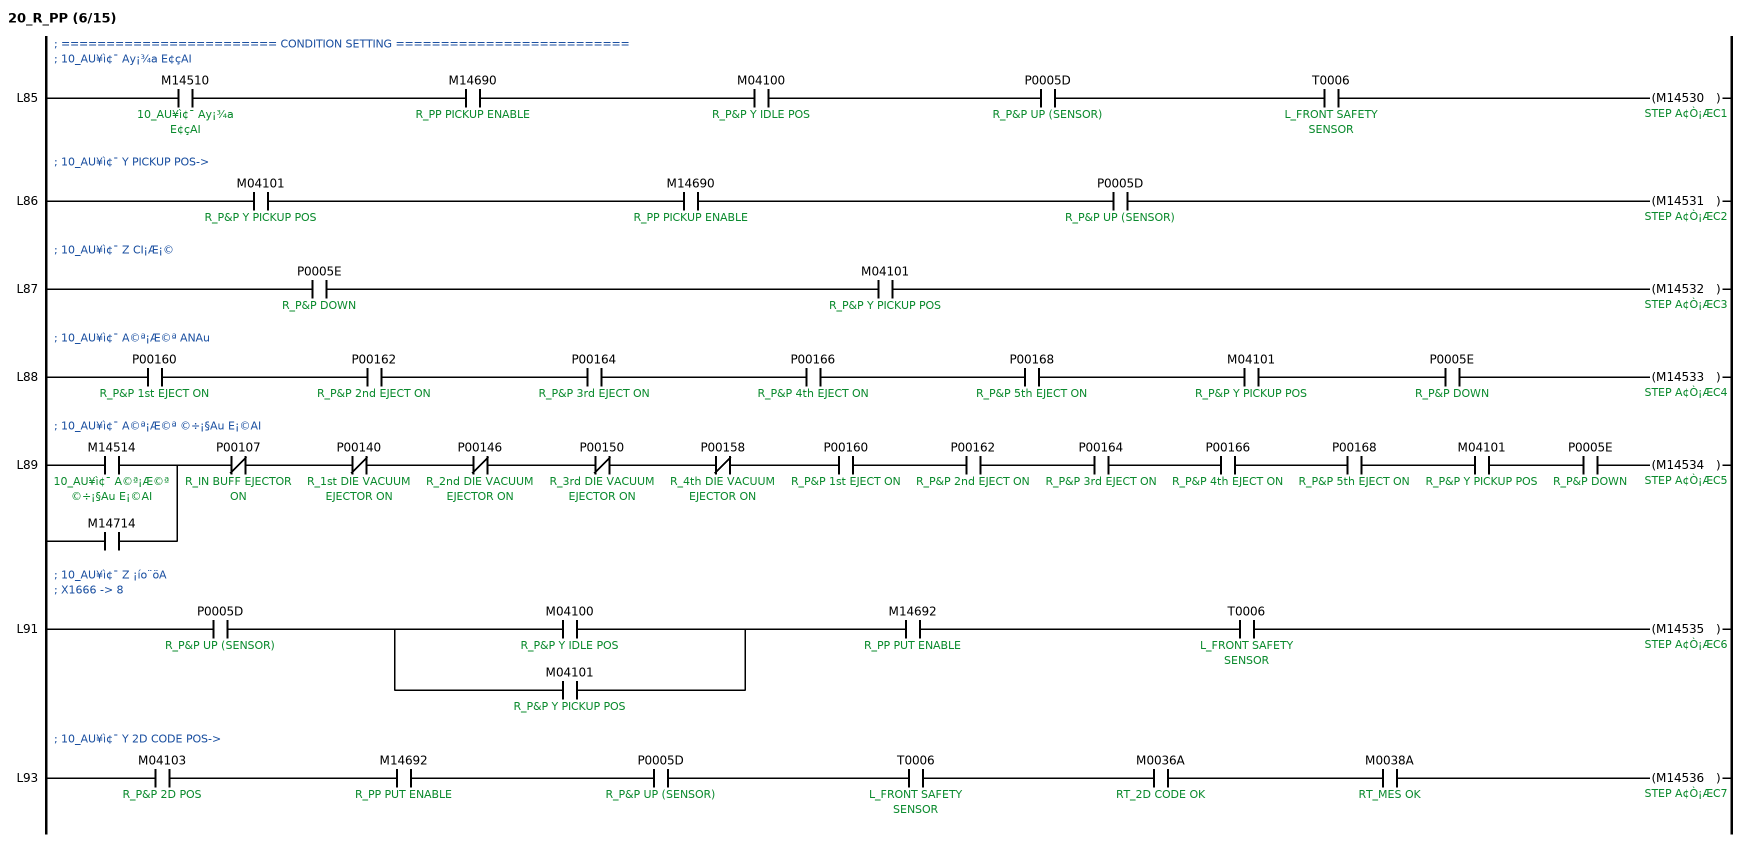
// ======================== CONDITION SETTING ==========================
; L85
LOAD      M14510	// 10_AU¥ì¢¯ Ay¡¾a E¢çAI
AND       M14690	// R_PP PICKUP ENABLE
AND       M04100	// R_P&P Y IDLE POS
AND       P0005D	// R_P&P UP (SENSOR)
AND       T0006	// L_FRONT SAFETY SENSOR
OUT       M14530	// STEP A¢Ò¡ÆC1
// output comment: 10_AU¥ì¢¯ Ay¡¾a E¢çAI
; L86
LOAD      M04101	// R_P&P Y PICKUP POS
AND       M14690	// R_PP PICKUP ENABLE
AND       P0005D	// R_P&P UP (SENSOR)
OUT       M14531	// STEP A¢Ò¡ÆC2
// output comment: 10_AU¥ì¢¯ Y PICKUP POS->
; L87
LOAD      P0005E	// R_P&P DOWN
AND       M04101	// R_P&P Y PICKUP POS
OUT       M14532	// STEP A¢Ò¡ÆC3
// output comment: 10_AU¥ì¢¯ Z CI¡Æ¡©
; L88
LOAD      P00160	// R_P&P 1st EJECT ON
AND       P00162	// R_P&P 2nd EJECT ON
AND       P00164	// R_P&P 3rd EJECT ON
AND       P00166	// R_P&P 4th EJECT ON
AND       P00168	// R_P&P 5th EJECT ON
AND       M04101	// R_P&P Y PICKUP POS
AND       P0005E	// R_P&P DOWN
OUT       M14533	// STEP A¢Ò¡ÆC4
// output comment: 10_AU¥ì¢¯ A©ª¡Æ©ª ANAu
; L89
LOAD      M14514	// 10_AU¥ì¢¯ A©ª¡Æ©ª ©÷¡§Au E¡©AI
OR        M14714
AND NOT   P00107	// R_IN BUFF EJECTOR ON
AND NOT   P00140	// R_1st DIE VACUUM EJECTOR ON
AND NOT   P00146	// R_2nd DIE VACUUM EJECTOR ON
AND NOT   P00150	// R_3rd DIE VACUUM EJECTOR ON
AND NOT   P00158	// R_4th DIE VACUUM EJECTOR ON
AND       P00160	// R_P&P 1st EJECT ON
AND       P00162	// R_P&P 2nd EJECT ON
AND       P00164	// R_P&P 3rd EJECT ON
AND       P00166	// R_P&P 4th EJECT ON
AND       P00168	// R_P&P 5th EJECT ON
AND       M04101	// R_P&P Y PICKUP POS
AND       P0005E	// R_P&P DOWN
OUT       M14534	// STEP A¢Ò¡ÆC5
// output comment: 10_AU¥ì¢¯ A©ª¡Æ©ª ©÷¡§Au E¡©AI
; L91
LOAD      P0005D	// R_P&P UP (SENSOR)
LOAD      M04100	// R_P&P Y IDLE POS
OR        M04101	// R_P&P Y PICKUP POS
AND LOAD
AND       M14692	// R_PP PUT ENABLE
AND       T0006	// L_FRONT SAFETY SENSOR
OUT       M14535	// STEP A¢Ò¡ÆC6
// output comment: 10_AU¥ì¢¯ Z ¡ío¨öA X1666 -> 8
; L93
LOAD      M04103	// R_P&P 2D POS
AND       M14692	// R_PP PUT ENABLE
AND       P0005D	// R_P&P UP (SENSOR)
AND       T0006	// L_FRONT SAFETY SENSOR
AND       M0036A	// RT_2D CODE OK
AND       M0038A	// RT_MES OK
OUT       M14536	// STEP A¢Ò¡ÆC7
// output comment: 10_AU¥ì¢¯ Y 2D CODE POS->

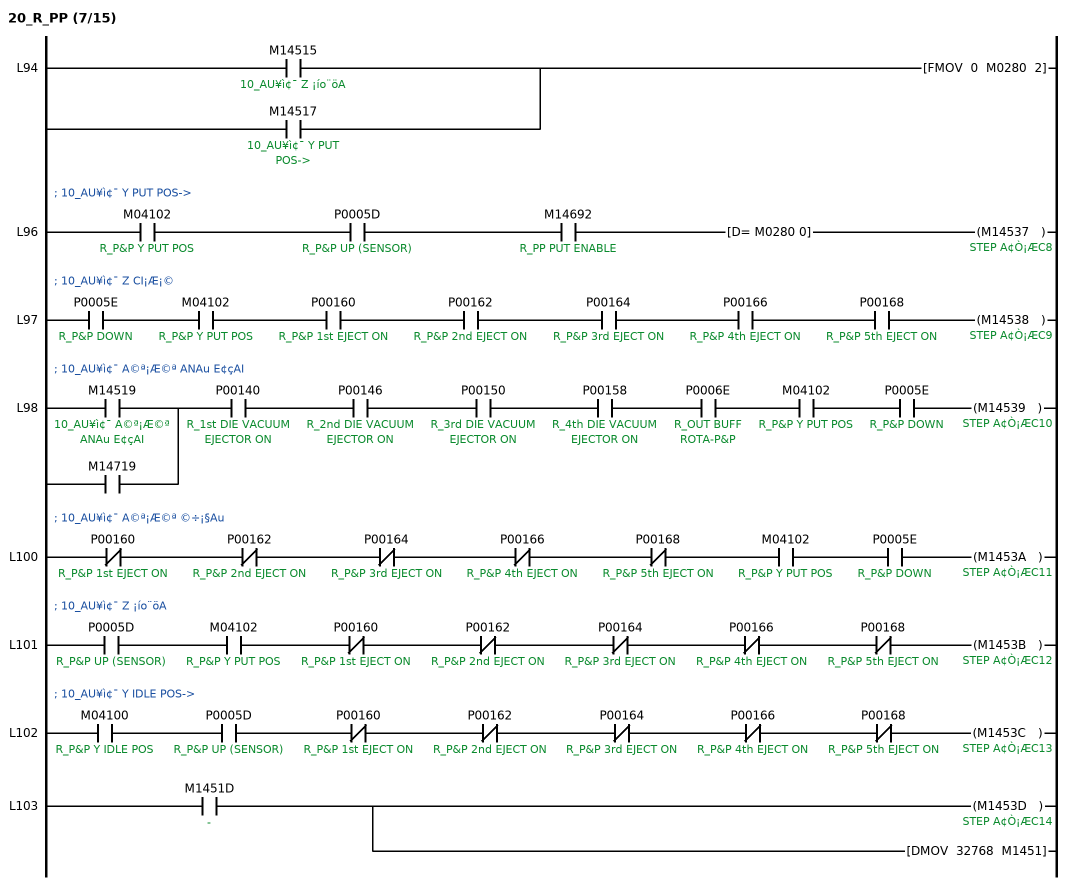
; L94
LOAD      M14515	// 10_AU¥ì¢¯ Z ¡ío¨öA
OR        M14517	// 10_AU¥ì¢¯ Y PUT POS->
FMOV      0 M0280 2
; L96
LOAD      M04102	// R_P&P Y PUT POS
AND       P0005D	// R_P&P UP (SENSOR)
AND       M14692	// R_PP PUT ENABLE
ANDD=     M0280 0
OUT       M14537	// STEP A¢Ò¡ÆC8
// output comment: 10_AU¥ì¢¯ Y PUT POS->
; L97
LOAD      P0005E	// R_P&P DOWN
AND       M04102	// R_P&P Y PUT POS
AND       P00160	// R_P&P 1st EJECT ON
AND       P00162	// R_P&P 2nd EJECT ON
AND       P00164	// R_P&P 3rd EJECT ON
AND       P00166	// R_P&P 4th EJECT ON
AND       P00168	// R_P&P 5th EJECT ON
OUT       M14538	// STEP A¢Ò¡ÆC9
// output comment: 10_AU¥ì¢¯ Z CI¡Æ¡©
; L98
LOAD      M14519	// 10_AU¥ì¢¯ A©ª¡Æ©ª ANAu E¢çAI
OR        M14719
AND       P00140	// R_1st DIE VACUUM EJECTOR ON
AND       P00146	// R_2nd DIE VACUUM EJECTOR ON
AND       P00150	// R_3rd DIE VACUUM EJECTOR ON
AND       P00158	// R_4th DIE VACUUM EJECTOR ON
AND       P0006E	// R_OUT BUFF ROTA-P&P
AND       M04102	// R_P&P Y PUT POS
AND       P0005E	// R_P&P DOWN
OUT       M14539	// STEP A¢Ò¡ÆC10
// output comment: 10_AU¥ì¢¯ A©ª¡Æ©ª ANAu E¢çAI
; L100
LOAD NOT  P00160	// R_P&P 1st EJECT ON
AND NOT   P00162	// R_P&P 2nd EJECT ON
AND NOT   P00164	// R_P&P 3rd EJECT ON
AND NOT   P00166	// R_P&P 4th EJECT ON
AND NOT   P00168	// R_P&P 5th EJECT ON
AND       M04102	// R_P&P Y PUT POS
AND       P0005E	// R_P&P DOWN
OUT       M1453A	// STEP A¢Ò¡ÆC11
// output comment: 10_AU¥ì¢¯ A©ª¡Æ©ª ©÷¡§Au
; L101
LOAD      P0005D	// R_P&P UP (SENSOR)
AND       M04102	// R_P&P Y PUT POS
AND NOT   P00160	// R_P&P 1st EJECT ON
AND NOT   P00162	// R_P&P 2nd EJECT ON
AND NOT   P00164	// R_P&P 3rd EJECT ON
AND NOT   P00166	// R_P&P 4th EJECT ON
AND NOT   P00168	// R_P&P 5th EJECT ON
OUT       M1453B	// STEP A¢Ò¡ÆC12
// output comment: 10_AU¥ì¢¯ Z ¡ío¨öA
; L102
LOAD      M04100	// R_P&P Y IDLE POS
AND       P0005D	// R_P&P UP (SENSOR)
AND NOT   P00160	// R_P&P 1st EJECT ON
AND NOT   P00162	// R_P&P 2nd EJECT ON
AND NOT   P00164	// R_P&P 3rd EJECT ON
AND NOT   P00166	// R_P&P 4th EJECT ON
AND NOT   P00168	// R_P&P 5th EJECT ON
OUT       M1453C	// STEP A¢Ò¡ÆC13
// output comment: 10_AU¥ì¢¯ Y IDLE POS->
; L103
LOAD      M1451D	// -
OUT       M1453D	// STEP A¢Ò¡ÆC14
DMOV      32768 M1451

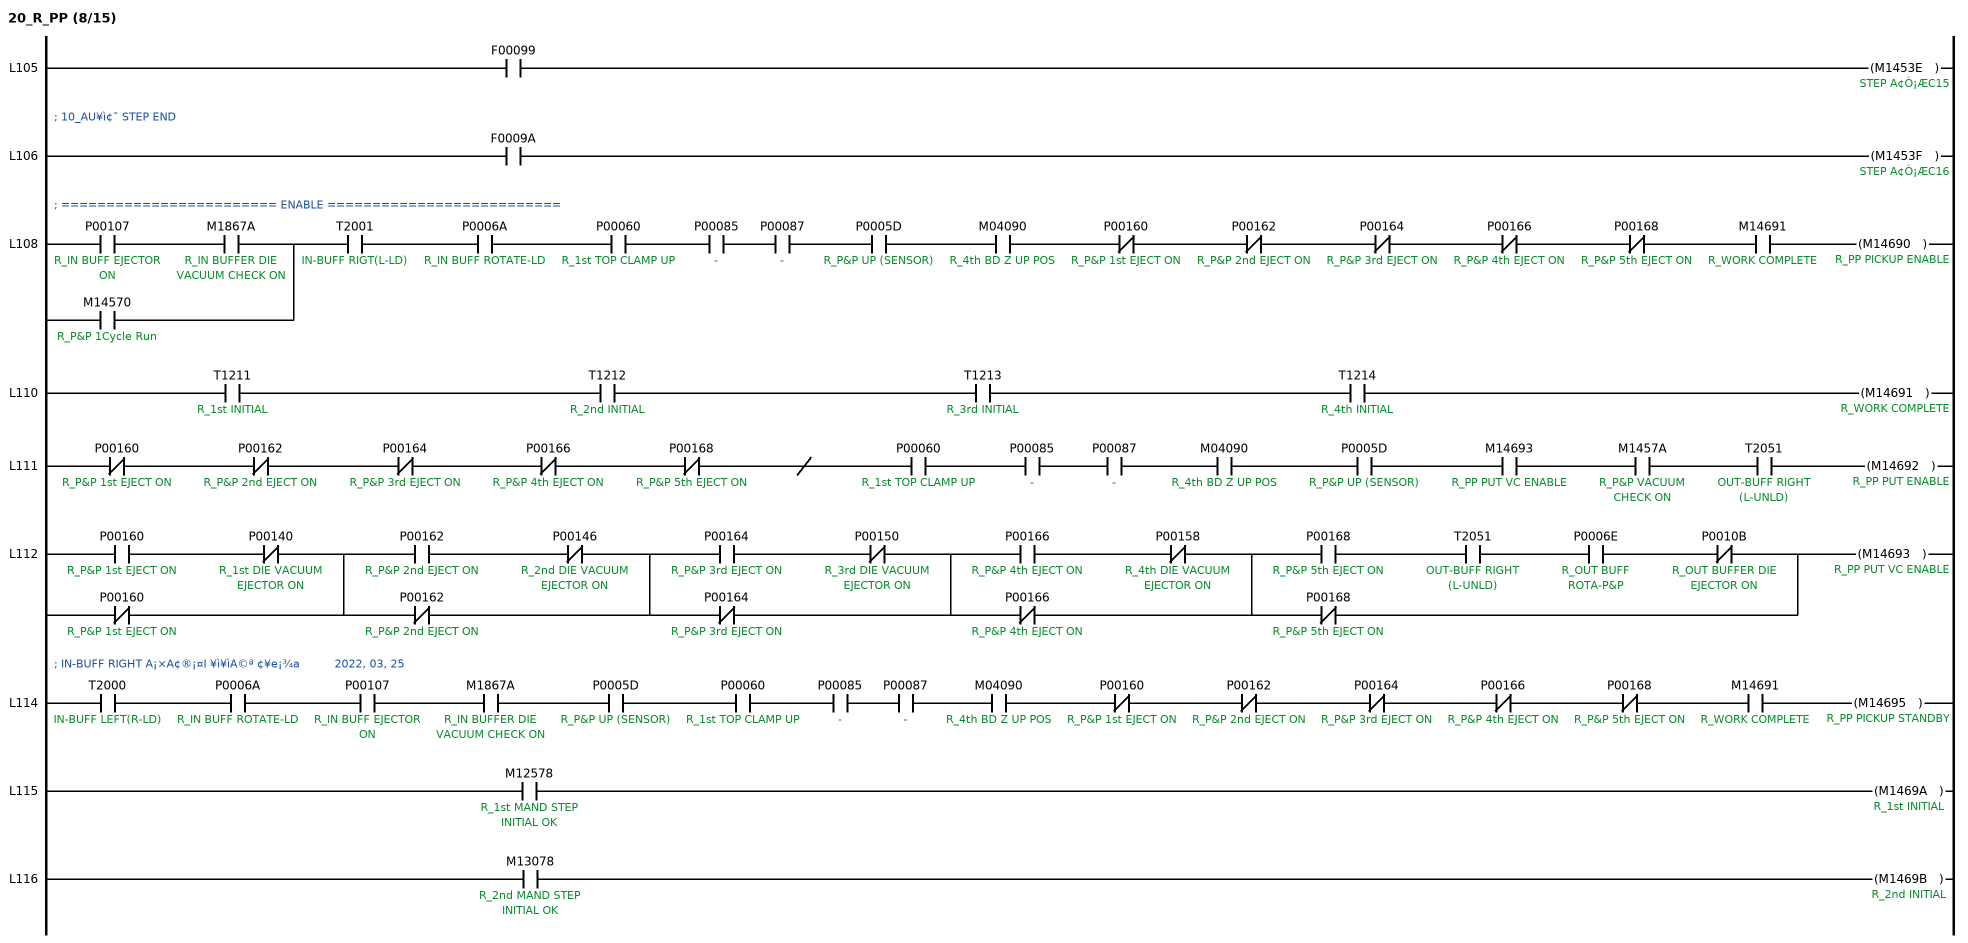
; L105
LOAD      F00099
OUT       M1453E	// STEP A¢Ò¡ÆC15
; L106
LOAD      F0009A
OUT       M1453F	// STEP A¢Ò¡ÆC16
// output comment: 10_AU¥ì¢¯ STEP END
// ======================== ENABLE ==========================
; L108
LOAD      P00107	// R_IN BUFF EJECTOR ON
AND       M1867A	// R_IN BUFFER DIE VACUUM CHECK ON
OR        M14570	// R_P&P 1Cycle Run
AND       T2001	// IN-BUFF RIGT(L-LD)
AND       P0006A	// R_IN BUFF ROTATE-LD
AND       P00060	// R_1st TOP CLAMP UP
AND       P00085	// -
AND       P00087	// -
AND       P0005D	// R_P&P UP (SENSOR)
AND       M04090	// R_4th BD Z UP POS
AND NOT   P00160	// R_P&P 1st EJECT ON
AND NOT   P00162	// R_P&P 2nd EJECT ON
AND NOT   P00164	// R_P&P 3rd EJECT ON
AND NOT   P00166	// R_P&P 4th EJECT ON
AND NOT   P00168	// R_P&P 5th EJECT ON
AND       M14691	// R_WORK COMPLETE
OUT       M14690	// R_PP PICKUP ENABLE
; L110
LOAD      T1211	// R_1st INITIAL
AND       T1212	// R_2nd INITIAL
AND       T1213	// R_3rd INITIAL
AND       T1214	// R_4th INITIAL
OUT       M14691	// R_WORK COMPLETE
; L111
LOAD NOT  P00160	// R_P&P 1st EJECT ON
AND NOT   P00162	// R_P&P 2nd EJECT ON
AND NOT   P00164	// R_P&P 3rd EJECT ON
AND NOT   P00166	// R_P&P 4th EJECT ON
AND NOT   P00168	// R_P&P 5th EJECT ON
NOT
AND       P00060	// R_1st TOP CLAMP UP
AND       P00085	// -
AND       P00087	// -
AND       M04090	// R_4th BD Z UP POS
AND       P0005D	// R_P&P UP (SENSOR)
AND       M14693	// R_PP PUT VC ENABLE
AND       M1457A	// R_P&P VACUUM CHECK ON
AND       T2051	// OUT-BUFF RIGHT (L-UNLD)
OUT       M14692	// R_PP PUT ENABLE
; L112
LOAD      P00160	// R_P&P 1st EJECT ON
AND NOT   P00140	// R_1st DIE VACUUM EJECTOR ON
OR NOT    P00160	// R_P&P 1st EJECT ON
LOAD      P00162	// R_P&P 2nd EJECT ON
AND NOT   P00146	// R_2nd DIE VACUUM EJECTOR ON
OR NOT    P00162	// R_P&P 2nd EJECT ON
AND LOAD
LOAD      P00164	// R_P&P 3rd EJECT ON
AND NOT   P00150	// R_3rd DIE VACUUM EJECTOR ON
OR NOT    P00164	// R_P&P 3rd EJECT ON
AND LOAD
LOAD      P00166	// R_P&P 4th EJECT ON
AND NOT   P00158	// R_4th DIE VACUUM EJECTOR ON
OR NOT    P00166	// R_P&P 4th EJECT ON
AND LOAD
LOAD      P00168	// R_P&P 5th EJECT ON
AND       T2051	// OUT-BUFF RIGHT (L-UNLD)
AND       P0006E	// R_OUT BUFF ROTA-P&P
AND NOT   P0010B	// R_OUT BUFFER DIE EJECTOR ON
OR NOT    P00168	// R_P&P 5th EJECT ON
AND LOAD
OUT       M14693	// R_PP PUT VC ENABLE
; L114
LOAD      T2000	// IN-BUFF LEFT(R-LD)
AND       P0006A	// R_IN BUFF ROTATE-LD
AND       P00107	// R_IN BUFF EJECTOR ON
AND       M1867A	// R_IN BUFFER DIE VACUUM CHECK ON
AND       P0005D	// R_P&P UP (SENSOR)
AND       P00060	// R_1st TOP CLAMP UP
AND       P00085	// -
AND       P00087	// -
AND       M04090	// R_4th BD Z UP POS
AND NOT   P00160	// R_P&P 1st EJECT ON
AND NOT   P00162	// R_P&P 2nd EJECT ON
AND NOT   P00164	// R_P&P 3rd EJECT ON
AND NOT   P00166	// R_P&P 4th EJECT ON
AND NOT   P00168	// R_P&P 5th EJECT ON
AND       M14691	// R_WORK COMPLETE
OUT       M14695	// R_PP PICKUP STANDBY
// output comment: IN-BUFF RIGHT A¡×A¢®¡¤I ¥ì¥ìA©ª ¢¥e¡¾a          2022, 03, 25
; L115
LOAD      M12578	// R_1st MAND STEP INITIAL OK
OUT       M1469A	// R_1st INITIAL
; L116
LOAD      M13078	// R_2nd MAND STEP INITIAL OK
OUT       M1469B	// R_2nd INITIAL

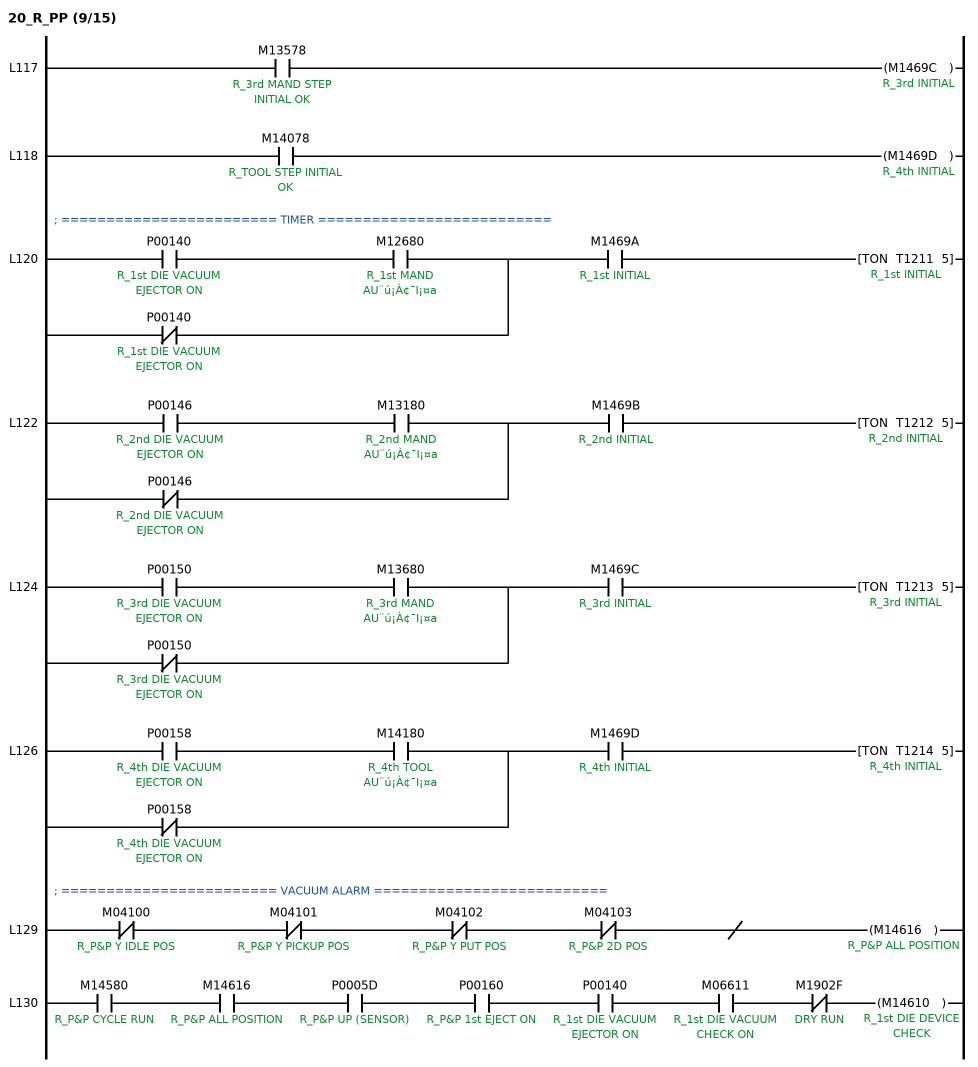
; L117
LOAD      M13578	// R_3rd MAND STEP INITIAL OK
OUT       M1469C	// R_3rd INITIAL
; L118
LOAD      M14078	// R_TOOL STEP INITIAL OK
OUT       M1469D	// R_4th INITIAL
// ======================== TIMER ==========================
; L120
LOAD      P00140	// R_1st DIE VACUUM EJECTOR ON
AND       M12680	// R_1st MAND AU¨ú¡À¢¯I¡¤a
OR NOT    P00140	// R_1st DIE VACUUM EJECTOR ON
AND       M1469A	// R_1st INITIAL
TON       T1211 5	// R_1st INITIAL
; L122
LOAD      P00146	// R_2nd DIE VACUUM EJECTOR ON
AND       M13180	// R_2nd MAND AU¨ú¡À¢¯I¡¤a
OR NOT    P00146	// R_2nd DIE VACUUM EJECTOR ON
AND       M1469B	// R_2nd INITIAL
TON       T1212 5	// R_2nd INITIAL
; L124
LOAD      P00150	// R_3rd DIE VACUUM EJECTOR ON
AND       M13680	// R_3rd MAND AU¨ú¡À¢¯I¡¤a
OR NOT    P00150	// R_3rd DIE VACUUM EJECTOR ON
AND       M1469C	// R_3rd INITIAL
TON       T1213 5	// R_3rd INITIAL
; L126
LOAD      P00158	// R_4th DIE VACUUM EJECTOR ON
AND       M14180	// R_4th TOOL AU¨ú¡À¢¯I¡¤a
OR NOT    P00158	// R_4th DIE VACUUM EJECTOR ON
AND       M1469D	// R_4th INITIAL
TON       T1214 5	// R_4th INITIAL
// ======================== VACUUM ALARM ==========================
; L129
LOAD NOT  M04100	// R_P&P Y IDLE POS
AND NOT   M04101	// R_P&P Y PICKUP POS
AND NOT   M04102	// R_P&P Y PUT POS
AND NOT   M04103	// R_P&P 2D POS
NOT
OUT       M14616	// R_P&P ALL POSITION
; L130
LOAD      M14580	// R_P&P CYCLE RUN
AND       M14616	// R_P&P ALL POSITION
AND       P0005D	// R_P&P UP (SENSOR)
AND       P00160	// R_P&P 1st EJECT ON
AND       P00140	// R_1st DIE VACUUM EJECTOR ON
AND       M06611	// R_1st DIE VACUUM CHECK ON
AND NOT   M1902F	// DRY RUN
OUT       M14610	// R_1st DIE DEVICE CHECK

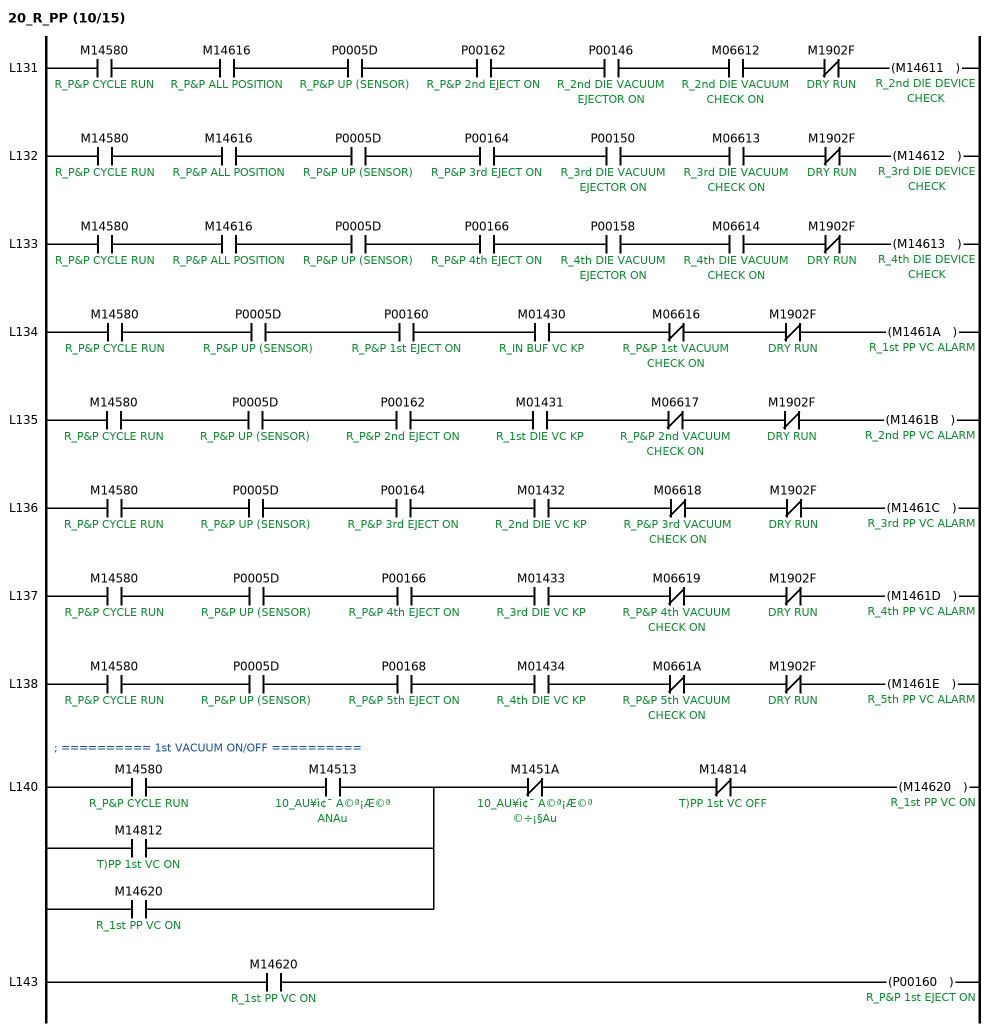
; L131
LOAD      M14580	// R_P&P CYCLE RUN
AND       M14616	// R_P&P ALL POSITION
AND       P0005D	// R_P&P UP (SENSOR)
AND       P00162	// R_P&P 2nd EJECT ON
AND       P00146	// R_2nd DIE VACUUM EJECTOR ON
AND       M06612	// R_2nd DIE VACUUM CHECK ON
AND NOT   M1902F	// DRY RUN
OUT       M14611	// R_2nd DIE DEVICE CHECK
; L132
LOAD      M14580	// R_P&P CYCLE RUN
AND       M14616	// R_P&P ALL POSITION
AND       P0005D	// R_P&P UP (SENSOR)
AND       P00164	// R_P&P 3rd EJECT ON
AND       P00150	// R_3rd DIE VACUUM EJECTOR ON
AND       M06613	// R_3rd DIE VACUUM CHECK ON
AND NOT   M1902F	// DRY RUN
OUT       M14612	// R_3rd DIE DEVICE CHECK
; L133
LOAD      M14580	// R_P&P CYCLE RUN
AND       M14616	// R_P&P ALL POSITION
AND       P0005D	// R_P&P UP (SENSOR)
AND       P00166	// R_P&P 4th EJECT ON
AND       P00158	// R_4th DIE VACUUM EJECTOR ON
AND       M06614	// R_4th DIE VACUUM CHECK ON
AND NOT   M1902F	// DRY RUN
OUT       M14613	// R_4th DIE DEVICE CHECK
; L134
LOAD      M14580	// R_P&P CYCLE RUN
AND       P0005D	// R_P&P UP (SENSOR)
AND       P00160	// R_P&P 1st EJECT ON
AND       M01430	// R_IN BUF VC KP
AND NOT   M06616	// R_P&P 1st VACUUM CHECK ON
AND NOT   M1902F	// DRY RUN
OUT       M1461A	// R_1st PP VC ALARM
; L135
LOAD      M14580	// R_P&P CYCLE RUN
AND       P0005D	// R_P&P UP (SENSOR)
AND       P00162	// R_P&P 2nd EJECT ON
AND       M01431	// R_1st DIE VC KP
AND NOT   M06617	// R_P&P 2nd VACUUM CHECK ON
AND NOT   M1902F	// DRY RUN
OUT       M1461B	// R_2nd PP VC ALARM
; L136
LOAD      M14580	// R_P&P CYCLE RUN
AND       P0005D	// R_P&P UP (SENSOR)
AND       P00164	// R_P&P 3rd EJECT ON
AND       M01432	// R_2nd DIE VC KP
AND NOT   M06618	// R_P&P 3rd VACUUM CHECK ON
AND NOT   M1902F	// DRY RUN
OUT       M1461C	// R_3rd PP VC ALARM
; L137
LOAD      M14580	// R_P&P CYCLE RUN
AND       P0005D	// R_P&P UP (SENSOR)
AND       P00166	// R_P&P 4th EJECT ON
AND       M01433	// R_3rd DIE VC KP
AND NOT   M06619	// R_P&P 4th VACUUM CHECK ON
AND NOT   M1902F	// DRY RUN
OUT       M1461D	// R_4th PP VC ALARM
; L138
LOAD      M14580	// R_P&P CYCLE RUN
AND       P0005D	// R_P&P UP (SENSOR)
AND       P00168	// R_P&P 5th EJECT ON
AND       M01434	// R_4th DIE VC KP
AND NOT   M0661A	// R_P&P 5th VACUUM CHECK ON
AND NOT   M1902F	// DRY RUN
OUT       M1461E	// R_5th PP VC ALARM
// ========== 1st VACUUM ON/OFF ==========
; L140
LOAD      M14580	// R_P&P CYCLE RUN
AND       M14513	// 10_AU¥ì¢¯ A©ª¡Æ©ª ANAu
OR        M14812	// T)PP 1st VC ON
OR        M14620	// R_1st PP VC ON
AND NOT   M1451A	// 10_AU¥ì¢¯ A©ª¡Æ©ª ©÷¡§Au
AND NOT   M14814	// T)PP 1st VC OFF
OUT       M14620	// R_1st PP VC ON
; L143
LOAD      M14620	// R_1st PP VC ON
OUT       P00160	// R_P&P 1st EJECT ON

